LIN {X 0,Y 714.172,Z 1021.651,A -85,B 0,C 180,E1 33366.658,E2 33366.658} C_VEL
LIN {X 0,Y 714.698,Z 1002.417,A -85,B 0,C 180,E1 33365.36,E2 33365.36} C_VEL
LIN {X 0,Y 715.219,Z 981.551,A -85,B 0,C 180,E1 33364.139,E2 33364.139} C_VEL
LIN {X 0,Y 715.786,Z 960.973,A -85,B 0,C 180,E1 33363.089,E2 33363.089} C_VEL
LIN {X 0,Y 716.314,Z 937.723,A -85,B 0,C 180,E1 33362.08,E2 33362.08} C_VEL
LIN {X 0,Y 716.774,Z 917.131,A -85,B 0,C 180,E1 33361.323,E2 33361.323} C_VEL
LIN {X 0,Y 717.276,Z 891.994,A -85,B 0,C 180,E1 33360.566,E2 33360.566} C_VEL
LIN {X 0,Y 717.596,Z 870.583,A -85,B 0,C 180,E1 33360.057,E2 33360.057} C_VEL
LIN {X 0,Y 717.997,Z 845.408,A -85,B 0,C 180,E1 33359.611,E2 33359.611} C_VEL
LIN {X 0,Y 718.258,Z 792.779,A -85,B 0,C 180,E1 33358.994,E2 33358.994} C_VEL
LIN {X 0,Y 719.244,Z 571.123,A -85,B 0,C 180,E1 33356.478,E2 33356.478} C_VEL
LIN {X 0,Y 719.679,Z 463.116,A -85,B 0,C 180,E1 33355.225,E2 33355.225} C_VEL
LIN {X 0,Y 717.181,Z 452.735,A -85,B 0,C 180,E1 33354.942,E2 33354.942} C_VEL
LIN {X 0,Y 717.903,Z 418.681,A -85,B 0,C 180,E1 33352.551,E2 33352.551} C_VEL
LIN {X 0,Y 712.298,Z 403.677,A -85,B 0,C 180,E1 33351.077,E2 33351.077} C_VEL
LIN {X 0,Y 712.228,Z 403.51,A -85,B 0,C 180,E1 33348.283,E2 33348.283} C_VEL
LIN {X 0,Y 712.278,Z 403.505,A -85,B 0,C 180,E1 33345.42,E2 33345.42} C_VEL
LIN {X 0,Y 712.238,Z 403.496,A -85,B 0,C 180,E1 33342.475,E2 33342.475} C_VEL
LIN {X 0,Y 712.277,Z 403.502,A -85,B 0,C 180,E1 33339.584,E2 33339.584} C_VEL
LIN {X 0,Y 712.255,Z 403.497,A -85,B 0,C 180,E1 33336.529,E2 33336.529} C_VEL
LIN {X 0,Y 712.277,Z 403.507,A -85,B 0,C 180,E1 33333.58,E2 33333.58} C_VEL
LIN {X 0,Y 712.263,Z 403.501,A -85,B 0,C 180,E1 33330.464,E2 33330.464} C_VEL
LIN {X 0,Y 712.279,Z 403.507,A -85,B 0,C 180,E1 33327.476,E2 33327.476} C_VEL
LIN {X 0,Y 712.269,Z 403.495,A -85,B 0,C 180,E1 33324.376,E2 33324.376} C_VEL
LIN {X 0,Y 712.281,Z 403.51,A -85,B 0,C 180,E1 33321.407,E2 33321.407} C_VEL
LIN {X 0,Y 712.275,Z 403.495,A -85,B 0,C 180,E1 33318.328,E2 33318.328} C_VEL
LIN {X 0,Y 712.28,Z 403.504,A -85,B 0,C 180,E1 33315.302,E2 33315.302} C_VEL
LIN {X 0,Y 712.28,Z 403.498,A -85,B 0,C 180,E1 33312.238,E2 33312.238} C_VEL
LIN {X 0,Y 712.272,Z 403.502,A -85,B 0,C 180,E1 33309.209,E2 33309.209} C_VEL
LIN {X 0,Y 712.276,Z 403.499,A -85,B 0,C 180,E1 33306.205,E2 33306.205} C_VEL
LIN {X 0,Y 712.268,Z 403.504,A -85,B 0,C 180,E1 33303.138,E2 33303.138} C_VEL
LIN {X 0,Y 712.267,Z 403.5,A -85,B 0,C 180,E1 33300.161,E2 33300.161} C_VEL
LIN {X 0,Y 712.261,Z 403.507,A -85,B 0,C 180,E1 33297.023,E2 33297.023} C_VEL
LIN {X 0,Y 712.255,Z 403.501,A -85,B 0,C 180,E1 33294.118,E2 33294.118} C_VEL
LIN {X 0,Y 712.265,Z 403.508,A -85,B 0,C 180,E1 33291.035,E2 33291.035} C_VEL
LIN {X 0,Y 712.233,Z 403.504,A -85,B 0,C 180,E1 33288.255,E2 33288.255} C_VEL
LIN {X 0,Y 712.281,Z 403.501,A -85,B 0,C 180,E1 33285.288,E2 33285.288} C_VEL
LIN {X 0,Y 712.223,Z 403.504,A -85,B 0,C 180,E1 33282.432,E2 33282.432} C_VEL
LIN {X 0,Y 712.253,Z 403.506,A -85,B 0,C 180,E1 33280.882,E2 33280.882} C_VEL
LIN {X 0,Y 711.211,Z 403.637,A -85,B 0,C 180,E1 33280.262,E2 33280.262} C_VEL
LIN {X 0,Y 704.791,Z 404.436,A -85,B 0,C 180,E1 33278.526,E2 33278.526} C_VEL
LIN {X 0,Y 704.281,Z 404.495,A -85,B 0,C 180,E1 33278.075,E2 33278.075} C_VEL
LIN {X 0,Y 704.342,Z 404.49,A -85,B 0,C 180,E1 33275.152,E2 33275.152} C_VEL
LIN {X 0,Y 704.273,Z 404.493,A -85,B 0,C 180,E1 33272.338,E2 33272.338} C_VEL
LIN {X 0,Y 704.287,Z 404.495,A -85,B 0,C 180,E1 33269.735,E2 33269.735} C_VEL
LIN {X 0,Y 704.284,Z 404.499,A -85,B 0,C 180,E1 33266.574,E2 33266.574} C_VEL
LIN {X 0,Y 704.259,Z 404.496,A -85,B 0,C 180,E1 33264,E2 33264} C_VEL
LIN {X 0,Y 704.331,Z 404.496,A -85,B 0,C 180,E1 33261.204,E2 33261.204} C_VEL
LIN {X 0,Y 704.254,Z 404.476,A -85,B 0,C 180,E1 33258.25,E2 33258.25} C_VEL
LIN {X 0,Y 704.248,Z 404.498,A -85,B 0,C 180,E1 33255.803,E2 33255.803} C_VEL
LIN {X 0,Y 704.323,Z 404.484,A -85,B 0,C 180,E1 33253.019,E2 33253.019} C_VEL
LIN {X 0,Y 704.244,Z 404.504,A -85,B 0,C 180,E1 33250.135,E2 33250.135} C_VEL
LIN {X 0,Y 704.232,Z 404.493,A -85,B 0,C 180,E1 33247.834,E2 33247.834} C_VEL
LIN {X 0,Y 704.252,Z 404.503,A -85,B 0,C 180,E1 33245.4,E2 33245.4} C_VEL
LIN {X 0,Y 704.289,Z 404.785,A -85,B 0,C 180,E1 33243.45,E2 33243.45} C_VEL
LIN {X 0,Y 707.485,Z 413.87,A -85,B 0,C 180,E1 33242.537,E2 33242.537} C_VEL
LIN {X 0,Y 712.329,Z 423.155,A -85,B 0,C 180,E1 33242.141,E2 33242.141} C_VEL
LIN {X 0,Y 713.266,Z 427.659,A -85,B 0,C 180,E1 33242.033,E2 33242.033} C_VEL
LIN {X 0,Y 711.801,Z 678.151,A -85,B 0,C 180,E1 33239.141,E2 33239.141} C_VEL
LIN {X 0,Y 711.089,Z 803.093,A -85,B 0,C 180,E1 33237.703,E2 33237.703} C_VEL
LIN {X 0,Y 710.685,Z 828.598,A -85,B 0,C 180,E1 33237.264,E2 33237.264} C_VEL
LIN {X 0,Y 710.266,Z 850.477,A -85,B 0,C 180,E1 33236.75,E2 33236.75} C_VEL
LIN {X 0,Y 709.752,Z 874.703,A -85,B 0,C 180,E1 33236.03,E2 33236.03} C_VEL
LIN {X 0,Y 709.172,Z 896.162,A -85,B 0,C 180,E1 33235.246,E2 33235.246} C_VEL
LIN {X 0,Y 708.554,Z 919.316,A -85,B 0,C 180,E1 33234.246,E2 33234.246} C_VEL
LIN {X 0,Y 707.886,Z 940.548,A -85,B 0,C 180,E1 33233.161,E2 33233.161} C_VEL
LIN {X 0,Y 707.238,Z 961.765,A -85,B 0,C 180,E1 33231.916,E2 33231.916} C_VEL
LIN {X 0,Y 706.634,Z 980.711,A -85,B 0,C 180,E1 33230.63,E2 33230.63} C_VEL
LIN {X 0,Y 706.061,Z 999.843,A -85,B 0,C 180,E1 33229.165,E2 33229.165} C_VEL
LIN {X 0,Y 705.555,Z 1017.001,A -85,B 0,C 180,E1 33227.654,E2 33227.654} C_VEL
LIN {X 0,Y 705.105,Z 1033.94,A -85,B 0,C 180,E1 33225.968,E2 33225.968} C_VEL
LIN {X 0,Y 704.748,Z 1047.913,A -85,B 0,C 180,E1 33224.376,E2 33224.376} C_VEL
LIN {X 0,Y 704.478,Z 1062.037,A -85,B 0,C 180,E1 33222.542,E2 33222.542} C_VEL
LIN {X 0,Y 704.26,Z 1073.543,A -85,B 0,C 180,E1 33220.802,E2 33220.802} C_VEL
LIN {X 0,Y 704.097,Z 1084.379,A -85,B 0,C 180,E1 33218.905,E2 33218.905} C_VEL
LIN {X 0,Y 703.993,Z 1092.895,A -85,B 0,C 180,E1 33217.098,E2 33217.098} C_VEL
LIN {X 0,Y 703.942,Z 1099.381,A -85,B 0,C 180,E1 33215.461,E2 33215.461} C_VEL
LIN {X 0,Y 703.9,Z 1105.808,A -85,B 0,C 180,E1 33213.42,E2 33213.42} C_VEL
LIN {X 0,Y 703.919,Z 1109.758,A -85,B 0,C 180,E1 33211.709,E2 33211.709} C_VEL
LIN {X 0,Y 703.913,Z 1112.752,A -85,B 0,C 180,E1 33209.837,E2 33209.837} C_VEL
LIN {X 0,Y 703.905,Z 1114.275,A -85,B 0,C 180,E1 33207.802,E2 33207.802} C_VEL
LIN {X 0,Y 703.9,Z 1114.27,A -85,B 0,C 180,E1 33206.09,E2 33206.09} C_VEL
LIN {X 0,Y 703.913,Z 1112.605,A -85,B 0,C 180,E1 33203.966,E2 33203.966} C_VEL
LIN {X 0,Y 703.92,Z 1109.684,A -85,B 0,C 180,E1 33202.162,E2 33202.162} C_VEL
LIN {X 0,Y 703.92,Z 1105.02,A -85,B 0,C 180,E1 33200.186,E2 33200.186} C_VEL
LIN {X 0,Y 703.938,Z 1098.76,A -85,B 0,C 180,E1 33198.28,E2 33198.28} C_VEL
LIN {X 0,Y 704.017,Z 1092.046,A -85,B 0,C 180,E1 33196.614,E2 33196.614} C_VEL
LIN {X 0,Y 704.116,Z 1082.18,A -85,B 0,C 180,E1 33194.6,E2 33194.6} C_VEL
LIN {X 0,Y 704.27,Z 1072.308,A -85,B 0,C 180,E1 33192.909,E2 33192.909} C_VEL
LIN {X 0,Y 704.521,Z 1059.625,A -85,B 0,C 180,E1 33191.034,E2 33191.034} C_VEL
LIN {X 0,Y 704.777,Z 1046.795,A -85,B 0,C 180,E1 33189.4,E2 33189.4} C_VEL
LIN {X 0,Y 705.159,Z 1031.359,A -85,B 0,C 180,E1 33187.665,E2 33187.665} C_VEL
LIN {X 0,Y 705.585,Z 1015.693,A -85,B 0,C 180,E1 33186.135,E2 33186.135} C_VEL
LIN {X 0,Y 706.113,Z 997.953,A -85,B 0,C 180,E1 33184.592,E2 33184.592} C_VEL
LIN {X 0,Y 706.658,Z 980.061,A -85,B 0,C 180,E1 33183.233,E2 33183.233} C_VEL
LIN {X 0,Y 707.287,Z 959.785,A -85,B 0,C 180,E1 33181.87,E2 33181.87} C_VEL
LIN {X 0,Y 707.92,Z 939.612,A -85,B 0,C 180,E1 33180.698,E2 33180.698} C_VEL
LIN {X 0,Y 708.605,Z 917.18,A -85,B 0,C 180,E1 33179.564,E2 33179.564} C_VEL
LIN {X 0,Y 709.184,Z 895.817,A -85,B 0,C 180,E1 33178.65,E2 33178.65} C_VEL
LIN {X 0,Y 709.806,Z 873.141,A -85,B 0,C 180,E1 33177.827,E2 33177.827} C_VEL
LIN {X 0,Y 710.287,Z 849.001,A -85,B 0,C 180,E1 33177.122,E2 33177.122} C_VEL
LIN {X 0,Y 710.771,Z 825.796,A -85,B 0,C 180,E1 33176.587,E2 33176.587} C_VEL
LIN {X 0,Y 711.1,Z 801.196,A -85,B 0,C 180,E1 33176.182,E2 33176.182} C_VEL
LIN {X 0,Y 712.566,Z 543.422,A -85,B 0,C 180,E1 33173.223,E2 33173.223} C_VEL
LIN {X 0,Y 713.097,Z 426.002,A -85,B 0,C 180,E1 33171.847,E2 33171.847} C_VEL
LIN {X 0,Y 711.559,Z 421.352,A -85,B 0,C 180,E1 33171.704,E2 33171.704} C_VEL
LIN {X 0,Y 707.344,Z 413.486,A -85,B 0,C 180,E1 33171.347,E2 33171.347} C_VEL
LIN {X 0,Y 704.271,Z 404.702,A -85,B 0,C 180,E1 33170.437,E2 33170.437} C_VEL
LIN {X 0,Y 704.236,Z 404.507,A -85,B 0,C 180,E1 33168.073,E2 33168.073} C_VEL
LIN {X 0,Y 704.276,Z 404.505,A -85,B 0,C 180,E1 33165.464,E2 33165.464} C_VEL
LIN {X 0,Y 704.262,Z 404.486,A -85,B 0,C 180,E1 33162.407,E2 33162.407} C_VEL
LIN {X 0,Y 704.249,Z 404.498,A -85,B 0,C 180,E1 33159.923,E2 33159.923} C_VEL
LIN {X 0,Y 704.28,Z 404.497,A -85,B 0,C 180,E1 33157.42,E2 33157.42} C_VEL
LIN {X 0,Y 704.275,Z 404.496,A -85,B 0,C 180,E1 33154.28,E2 33154.28} C_VEL
LIN {X 0,Y 704.262,Z 404.497,A -85,B 0,C 180,E1 33151.74,E2 33151.74} C_VEL
LIN {X 0,Y 704.339,Z 404.476,A -85,B 0,C 180,E1 33148.953,E2 33148.953} C_VEL
LIN {X 0,Y 704.277,Z 404.496,A -85,B 0,C 180,E1 33146.012,E2 33146.012} C_VEL
LIN {X 0,Y 704.282,Z 404.493,A -85,B 0,C 180,E1 33143.424,E2 33143.424} C_VEL
LIN {X 0,Y 704.337,Z 404.487,A -85,B 0,C 180,E1 33140.44,E2 33140.44} C_VEL
LIN {X 0,Y 704.281,Z 404.497,A -85,B 0,C 180,E1 33137.602,E2 33137.602} C_VEL
LIN {X 0,Y 704.346,Z 404.494,A -85,B 0,C 180,E1 33134.805,E2 33134.805} C_VEL
LIN {X 0,Y 704.296,Z 404.488,A -85,B 0,C 180,E1 33131.797,E2 33131.797} C_VEL
LIN {X 0,Y 704.321,Z 404.499,A -85,B 0,C 180,E1 33128.984,E2 33128.984} C_VEL
LIN {X 0,Y 704.314,Z 404.488,A -85,B 0,C 180,E1 33125.867,E2 33125.867} C_VEL
LIN {X 0,Y 704.324,Z 404.498,A -85,B 0,C 180,E1 33122.93,E2 33122.93} C_VEL
LIN {X 0,Y 704.327,Z 404.489,A -85,B 0,C 180,E1 33119.837,E2 33119.837} C_VEL
LIN {X 0,Y 704.33,Z 404.491,A -85,B 0,C 180,E1 33116.826,E2 33116.826} C_VEL
LIN {X 0,Y 704.331,Z 404.486,A -85,B 0,C 180,E1 33113.724,E2 33113.724} C_VEL
LIN {X 0,Y 704.337,Z 404.497,A -85,B 0,C 180,E1 33110.686,E2 33110.686} C_VEL
LIN {X 0,Y 704.334,Z 404.482,A -85,B 0,C 180,E1 33107.609,E2 33107.609} C_VEL
LIN {X 0,Y 704.34,Z 404.494,A -85,B 0,C 180,E1 33104.521,E2 33104.521} C_VEL
LIN {X 0,Y 704.334,Z 404.489,A -85,B 0,C 180,E1 33101.458,E2 33101.458} C_VEL
LIN {X 0,Y 704.333,Z 404.488,A -85,B 0,C 180,E1 33098.413,E2 33098.413} C_VEL
LIN {X 0,Y 704.342,Z 404.488,A -85,B 0,C 180,E1 33095.421,E2 33095.421} C_VEL
LIN {X 0,Y 704.328,Z 404.495,A -85,B 0,C 180,E1 33092.34,E2 33092.34} C_VEL
LIN {X 0,Y 704.34,Z 404.485,A -85,B 0,C 180,E1 33089.349,E2 33089.349} C_VEL
LIN {X 0,Y 704.327,Z 404.497,A -85,B 0,C 180,E1 33086.284,E2 33086.284} C_VEL
LIN {X 0,Y 704.332,Z 404.489,A -85,B 0,C 180,E1 33083.297,E2 33083.297} C_VEL
LIN {X 0,Y 704.317,Z 404.497,A -85,B 0,C 180,E1 33080.178,E2 33080.178} C_VEL
LIN {X 0,Y 704.318,Z 404.486,A -85,B 0,C 180,E1 33077.266,E2 33077.266} C_VEL
LIN {X 0,Y 704.321,Z 404.495,A -85,B 0,C 180,E1 33074.191,E2 33074.191} C_VEL
LIN {X 0,Y 704.296,Z 404.499,A -85,B 0,C 180,E1 33071.421,E2 33071.421} C_VEL
LIN {X 0,Y 704.325,Z 404.718,A -85,B 0,C 180,E1 33069.336,E2 33069.336} C_VEL
LIN {X 0,Y 710.956,Z 422.229,A -85,B 0,C 180,E1 33067.617,E2 33067.617} C_VEL
LIN {X 0,Y 710.223,Z 453.298,A -85,B 0,C 180,E1 33065.43,E2 33065.43} C_VEL
LIN {X 0,Y 713.265,Z 466.404,A -85,B 0,C 180,E1 33065.094,E2 33065.094} C_VEL
LIN {X 0,Y 711.805,Z 716.052,A -85,B 0,C 180,E1 33062.21,E2 33062.21} C_VEL
LIN {X 0,Y 711.1,Z 842.987,A -85,B 0,C 180,E1 33060.749,E2 33060.749} C_VEL
LIN {X 0,Y 710.684,Z 868.493,A -85,B 0,C 180,E1 33060.311,E2 33060.311} C_VEL
LIN {X 0,Y 710.261,Z 890.337,A -85,B 0,C 180,E1 33059.798,E2 33059.798} C_VEL
LIN {X 0,Y 709.761,Z 914.559,A -85,B 0,C 180,E1 33059.08,E2 33059.08} C_VEL
LIN {X 0,Y 709.162,Z 936.485,A -85,B 0,C 180,E1 33058.278,E2 33058.278} C_VEL
LIN {X 0,Y 708.561,Z 959.167,A -85,B 0,C 180,E1 33057.299,E2 33057.299} C_VEL
LIN {X 0,Y 707.877,Z 980.757,A -85,B 0,C 180,E1 33056.194,E2 33056.194} C_VEL
LIN {X 0,Y 707.237,Z 1001.75,A -85,B 0,C 180,E1 33054.962,E2 33054.962} C_VEL
LIN {X 0,Y 706.629,Z 1021.05,A -85,B 0,C 180,E1 33053.651,E2 33053.651} C_VEL
LIN {X 0,Y 706.064,Z 1039.761,A -85,B 0,C 180,E1 33052.217,E2 33052.217} C_VEL
LIN {X 0,Y 705.561,Z 1056.796,A -85,B 0,C 180,E1 33050.719,E2 33050.719} C_VEL
LIN {X 0,Y 705.139,Z 1072.966,A -85,B 0,C 180,E1 33049.121,E2 33049.121} C_VEL
LIN {X 0,Y 704.764,Z 1087.223,A -85,B 0,C 180,E1 33047.504,E2 33047.504} C_VEL
LIN {X 0,Y 704.491,Z 1101.06,A -85,B 0,C 180,E1 33045.729,E2 33045.729} C_VEL
LIN {X 0,Y 704.27,Z 1112.797,A -85,B 0,C 180,E1 33043.967,E2 33043.967} C_VEL
LIN {X 0,Y 704.122,Z 1122.947,A -85,B 0,C 180,E1 33042.215,E2 33042.215} C_VEL
LIN {X 0,Y 704.014,Z 1132.538,A -85,B 0,C 180,E1 33040.226,E2 33040.226} C_VEL
LIN {X 0,Y 703.947,Z 1139.12,A -85,B 0,C 180,E1 33038.577,E2 33038.577} C_VEL
LIN {X 0,Y 703.922,Z 1145.451,A -85,B 0,C 180,E1 33036.607,E2 33036.607} C_VEL
LIN {X 0,Y 703.911,Z 1149.814,A -85,B 0,C 180,E1 33034.726,E2 33034.726} C_VEL
LIN {X 0,Y 703.882,Z 1152.685,A -85,B 0,C 180,E1 33032.931,E2 33032.931} C_VEL
LIN {X 0,Y 703.892,Z 1154.262,A -85,B 0,C 180,E1 33030.895,E2 33030.895} C_VEL
LIN {X 0,Y 703.884,Z 1154.306,A -85,B 0,C 180,E1 33029.267,E2 33029.267} C_VEL
LIN {X 0,Y 703.886,Z 1153.017,A -85,B 0,C 180,E1 33027.313,E2 33027.313} C_VEL
LIN {X 0,Y 703.916,Z 1149.972,A -85,B 0,C 180,E1 33025.356,E2 33025.356} C_VEL
LIN {X 0,Y 703.921,Z 1145.864,A -85,B 0,C 180,E1 33023.557,E2 33023.557} C_VEL
LIN {X 0,Y 703.948,Z 1139.423,A -85,B 0,C 180,E1 33021.505,E2 33021.505} C_VEL
LIN {X 0,Y 704.009,Z 1132.739,A -85,B 0,C 180,E1 33019.821,E2 33019.821} C_VEL
LIN {X 0,Y 704.116,Z 1123.406,A -85,B 0,C 180,E1 33017.868,E2 33017.868} C_VEL
LIN {X 0,Y 704.262,Z 1113.319,A -85,B 0,C 180,E1 33016.117,E2 33016.117} C_VEL
LIN {X 0,Y 704.473,Z 1101.643,A -85,B 0,C 180,E1 33014.355,E2 33014.355} C_VEL
LIN {X 0,Y 704.746,Z 1087.93,A -85,B 0,C 180,E1 33012.58,E2 33012.58} C_VEL
LIN {X 0,Y 705.118,Z 1073.742,A -85,B 0,C 180,E1 33010.965,E2 33010.965} C_VEL
LIN {X 0,Y 705.542,Z 1057.389,A -85,B 0,C 180,E1 33009.336,E2 33009.336} C_VEL
LIN {X 0,Y 706.035,Z 1040.55,A -85,B 0,C 180,E1 33007.85,E2 33007.85} C_VEL
LIN {X 0,Y 706.609,Z 1021.653,A -85,B 0,C 180,E1 33006.393,E2 33006.393} C_VEL
LIN {X 0,Y 707.213,Z 1002.413,A -85,B 0,C 180,E1 33005.082,E2 33005.082} C_VEL
LIN {X 0,Y 707.847,Z 981.555,A -85,B 0,C 180,E1 33003.85,E2 33003.85} C_VEL
LIN {X 0,Y 708.499,Z 960.969,A -85,B 0,C 180,E1 33002.79,E2 33002.79} C_VEL
LIN {X 0,Y 709.128,Z 937.608,A -85,B 0,C 180,E1 33001.766,E2 33001.766} C_VEL
LIN {X 0,Y 709.672,Z 917.128,A -85,B 0,C 180,E1 33001.008,E2 33001.008} C_VEL
LIN {X 0,Y 710.244,Z 892.062,A -85,B 0,C 180,E1 33000.247,E2 33000.247} C_VEL
LIN {X 0,Y 710.629,Z 870.451,A -85,B 0,C 180,E1 32999.73,E2 32999.73} C_VEL
LIN {X 0,Y 711.088,Z 845.088,A -85,B 0,C 180,E1 32999.28,E2 32999.28} C_VEL
LIN {X 0,Y 711.421,Z 788.58,A -85,B 0,C 180,E1 32998.614,E2 32998.614} C_VEL
LIN {X 0,Y 712.582,Z 568.705,A -85,B 0,C 180,E1 32996.094,E2 32996.094} C_VEL
LIN {X 0,Y 713.087,Z 464.856,A -85,B 0,C 180,E1 32994.878,E2 32994.878} C_VEL
LIN {X 0,Y 710.17,Z 452.741,A -85,B 0,C 180,E1 32994.544,E2 32994.544} C_VEL
LIN {X 0,Y 710.885,Z 422.01,A -85,B 0,C 180,E1 32992.362,E2 32992.362} C_VEL
LIN {X 0,Y 704.321,Z 404.695,A -85,B 0,C 180,E1 32990.653,E2 32990.653} C_VEL
LIN {X 0,Y 704.3,Z 404.496,A -85,B 0,C 180,E1 32988.035,E2 32988.035} C_VEL
LIN {X 0,Y 704.34,Z 404.492,A -85,B 0,C 180,E1 32984.989,E2 32984.989} C_VEL
LIN {X 0,Y 704.3,Z 404.478,A -85,B 0,C 180,E1 32982.075,E2 32982.075} C_VEL
LIN {X 0,Y 704.336,Z 404.495,A -85,B 0,C 180,E1 32979.178,E2 32979.178} C_VEL
LIN {X 0,Y 704.303,Z 404.489,A -85,B 0,C 180,E1 32976.256,E2 32976.256} C_VEL
LIN {X 0,Y 704.339,Z 404.492,A -85,B 0,C 180,E1 32973.411,E2 32973.411} C_VEL
LIN {X 0,Y 704.318,Z 404.492,A -85,B 0,C 180,E1 32970.358,E2 32970.358} C_VEL
LIN {X 0,Y 704.338,Z 404.497,A -85,B 0,C 180,E1 32967.384,E2 32967.384} C_VEL
LIN {X 0,Y 704.325,Z 404.484,A -85,B 0,C 180,E1 32964.312,E2 32964.312} C_VEL
LIN {X 0,Y 704.337,Z 404.497,A -85,B 0,C 180,E1 32961.311,E2 32961.311} C_VEL
LIN {X 0,Y 704.332,Z 404.485,A -85,B 0,C 180,E1 32958.243,E2 32958.243} C_VEL
LIN {X 0,Y 704.333,Z 404.492,A -85,B 0,C 180,E1 32955.226,E2 32955.226} C_VEL
LIN {X 0,Y 704.339,Z 404.487,A -85,B 0,C 180,E1 32952.212,E2 32952.212} C_VEL
LIN {X 0,Y 704.329,Z 404.49,A -85,B 0,C 180,E1 32949.149,E2 32949.149} C_VEL
LIN {X 0,Y 704.342,Z 404.488,A -85,B 0,C 180,E1 32946.112,E2 32946.112} C_VEL
LIN {X 0,Y 704.319,Z 404.493,A -85,B 0,C 180,E1 32943.011,E2 32943.011} C_VEL
LIN {X 0,Y 704.347,Z 404.488,A -85,B 0,C 180,E1 32940,E2 32940} C_VEL
LIN {X 0,Y 704.312,Z 404.494,A -85,B 0,C 180,E1 32936.908,E2 32936.908} C_VEL
LIN {X 0,Y 704.332,Z 404.489,A -85,B 0,C 180,E1 32933.97,E2 32933.97} C_VEL
LIN {X 0,Y 704.315,Z 404.497,A -85,B 0,C 180,E1 32930.933,E2 32930.933} C_VEL
LIN {X 0,Y 704.302,Z 404.491,A -85,B 0,C 180,E1 32928.12,E2 32928.12} C_VEL
LIN {X 0,Y 704.338,Z 404.494,A -85,B 0,C 180,E1 32925.111,E2 32925.111} C_VEL
LIN {X 0,Y 704.284,Z 404.492,A -85,B 0,C 180,E1 32922.296,E2 32922.296} C_VEL
LIN {X 0,Y 704.343,Z 404.49,A -85,B 0,C 180,E1 32919.386,E2 32919.386} C_VEL
LIN {X 0,Y 704.281,Z 404.495,A -85,B 0,C 180,E1 32918.075,E2 32918.075} C_VEL
LIN {X 0,Y 703.324,Z 404.621,A -85,B 0,C 180,E1 32917.448,E2 32917.448} C_VEL
LIN {X 0,Y 696.939,Z 405.403,A -85,B 0,C 180,E1 32915.692,E2 32915.692} C_VEL
LIN {X 0,Y 696.404,Z 405.475,A -85,B 0,C 180,E1 32915.236,E2 32915.236} C_VEL
LIN {X 0,Y 696.335,Z 405.482,A -85,B 0,C 180,E1 32912.367,E2 32912.367} C_VEL
LIN {X 0,Y 696.349,Z 405.484,A -85,B 0,C 180,E1 32909.735,E2 32909.735} C_VEL
LIN {X 0,Y 696.353,Z 405.488,A -85,B 0,C 180,E1 32906.636,E2 32906.636} C_VEL
LIN {X 0,Y 696.319,Z 405.485,A -85,B 0,C 180,E1 32904.033,E2 32904.033} C_VEL
LIN {X 0,Y 696.37,Z 405.486,A -85,B 0,C 180,E1 32901.347,E2 32901.347} C_VEL
LIN {X 0,Y 696.32,Z 405.462,A -85,B 0,C 180,E1 32898.329,E2 32898.329} C_VEL
LIN {X 0,Y 696.308,Z 405.487,A -85,B 0,C 180,E1 32895.856,E2 32895.856} C_VEL
LIN {X 0,Y 696.37,Z 405.474,A -85,B 0,C 180,E1 32893.116,E2 32893.116} C_VEL
LIN {X 0,Y 696.306,Z 405.493,A -85,B 0,C 180,E1 32890.148,E2 32890.148} C_VEL
LIN {X 0,Y 696.294,Z 405.481,A -85,B 0,C 180,E1 32887.82,E2 32887.82} C_VEL
LIN {X 0,Y 696.327,Z 405.486,A -85,B 0,C 180,E1 32885.258,E2 32885.258} C_VEL
LIN {X 0,Y 696.337,Z 405.747,A -85,B 0,C 180,E1 32883.883,E2 32883.883} C_VEL
LIN {X 0,Y 699.249,Z 413.816,A -85,B 0,C 180,E1 32883.026,E2 32883.026} C_VEL
LIN {X 0,Y 706.323,Z 427.111,A -85,B 0,C 180,E1 32882.437,E2 32882.437} C_VEL
LIN {X 0,Y 706.698,Z 430.076,A -85,B 0,C 180,E1 32882.379,E2 32882.379} C_VEL
LIN {X 0,Y 705.014,Z 680.25,A -85,B 0,C 180,E1 32879.464,E2 32879.464} C_VEL
LIN {X 0,Y 704.203,Z 803.228,A -85,B 0,C 180,E1 32878.035,E2 32878.035} C_VEL
LIN {X 0,Y 703.751,Z 828.68,A -85,B 0,C 180,E1 32877.593,E2 32877.593} C_VEL
LIN {X 0,Y 703.261,Z 850.534,A -85,B 0,C 180,E1 32877.076,E2 32877.076} C_VEL
LIN {X 0,Y 702.637,Z 875.784,A -85,B 0,C 180,E1 32876.314,E2 32876.314} C_VEL
LIN {X 0,Y 702.023,Z 896.009,A -85,B 0,C 180,E1 32875.567,E2 32875.567} C_VEL
LIN {X 0,Y 701.322,Z 918.305,A -85,B 0,C 180,E1 32874.602,E2 32874.602} C_VEL
LIN {X 0,Y 700.544,Z 940.37,A -85,B 0,C 180,E1 32873.467,E2 32873.467} C_VEL
LIN {X 0,Y 699.805,Z 961.02,A -85,B 0,C 180,E1 32872.249,E2 32872.249} C_VEL
LIN {X 0,Y 699.096,Z 980.58,A -85,B 0,C 180,E1 32870.911,E2 32870.911} C_VEL
LIN {X 0,Y 698.424,Z 999.594,A -85,B 0,C 180,E1 32869.442,E2 32869.442} C_VEL
LIN {X 0,Y 697.842,Z 1016.566,A -85,B 0,C 180,E1 32867.935,E2 32867.935} C_VEL
LIN {X 0,Y 697.336,Z 1032.748,A -85,B 0,C 180,E1 32866.322,E2 32866.322} C_VEL
LIN {X 0,Y 696.914,Z 1047.521,A -85,B 0,C 180,E1 32864.626,E2 32864.626} C_VEL
LIN {X 0,Y 696.6,Z 1061.144,A -85,B 0,C 180,E1 32862.855,E2 32862.855} C_VEL
LIN {X 0,Y 696.32,Z 1073.254,A -85,B 0,C 180,E1 32861.01,E2 32861.01} C_VEL
LIN {X 0,Y 696.137,Z 1083.703,A -85,B 0,C 180,E1 32859.174,E2 32859.174} C_VEL
LIN {X 0,Y 696.026,Z 1092.695,A -85,B 0,C 180,E1 32857.263,E2 32857.263} C_VEL
LIN {X 0,Y 695.948,Z 1099.51,A -85,B 0,C 180,E1 32855.524,E2 32855.524} C_VEL
LIN {X 0,Y 695.903,Z 1105.896,A -85,B 0,C 180,E1 32853.46,E2 32853.46} C_VEL
LIN {X 0,Y 695.92,Z 1109.826,A -85,B 0,C 180,E1 32851.729,E2 32851.729} C_VEL
LIN {X 0,Y 695.909,Z 1112.912,A -85,B 0,C 180,E1 32849.753,E2 32849.753} C_VEL
LIN {X 0,Y 695.903,Z 1114.284,A -85,B 0,C 180,E1 32847.777,E2 32847.777} C_VEL
LIN {X 0,Y 695.904,Z 1114.261,A -85,B 0,C 180,E1 32846.045,E2 32846.045} C_VEL
LIN {X 0,Y 695.918,Z 1112.558,A -85,B 0,C 180,E1 32843.897,E2 32843.897} C_VEL
LIN {X 0,Y 695.919,Z 1109.617,A -85,B 0,C 180,E1 32842.072,E2 32842.072} C_VEL
LIN {X 0,Y 695.933,Z 1104.911,A -85,B 0,C 180,E1 32840.072,E2 32840.072} C_VEL
LIN {X 0,Y 695.947,Z 1098.935,A -85,B 0,C 180,E1 32838.228,E2 32838.228} C_VEL
LIN {X 0,Y 696.039,Z 1092.251,A -85,B 0,C 180,E1 32836.543,E2 32836.543} C_VEL
LIN {X 0,Y 696.155,Z 1082.443,A -85,B 0,C 180,E1 32834.505,E2 32834.505} C_VEL
LIN {X 0,Y 696.329,Z 1072.607,A -85,B 0,C 180,E1 32832.794,E2 32832.794} C_VEL
LIN {X 0,Y 696.609,Z 1059.988,A -85,B 0,C 180,E1 32830.897,E2 32830.897} C_VEL
LIN {X 0,Y 696.923,Z 1047.201,A -85,B 0,C 180,E1 32829.245,E2 32829.245} C_VEL
LIN {X 0,Y 697.36,Z 1031.842,A -85,B 0,C 180,E1 32827.491,E2 32827.491} C_VEL
LIN {X 0,Y 697.873,Z 1015.528,A -85,B 0,C 180,E1 32825.878,E2 32825.878} C_VEL
LIN {X 0,Y 698.487,Z 997.829,A -85,B 0,C 180,E1 32824.324,E2 32824.324} C_VEL
LIN {X 0,Y 699.119,Z 979.873,A -85,B 0,C 180,E1 32822.947,E2 32822.947} C_VEL
LIN {X 0,Y 699.84,Z 959.882,A -85,B 0,C 180,E1 32821.59,E2 32821.59} C_VEL
LIN {X 0,Y 700.568,Z 939.715,A -85,B 0,C 180,E1 32820.407,E2 32820.407} C_VEL
LIN {X 0,Y 701.338,Z 917.756,A -85,B 0,C 180,E1 32819.282,E2 32819.282} C_VEL
LIN {X 0,Y 702.025,Z 895.969,A -85,B 0,C 180,E1 32818.342,E2 32818.342} C_VEL
LIN {X 0,Y 702.693,Z 874.286,A -85,B 0,C 180,E1 32817.545,E2 32817.545} C_VEL
LIN {X 0,Y 703.275,Z 849.84,A -85,B 0,C 180,E1 32816.816,E2 32816.816} C_VEL
LIN {X 0,Y 703.787,Z 827.578,A -85,B 0,C 180,E1 32816.294,E2 32816.294} C_VEL
LIN {X 0,Y 704.21,Z 802.207,A -85,B 0,C 180,E1 32815.861,E2 32815.861} C_VEL
LIN {X 0,Y 705.874,Z 548.474,A -85,B 0,C 180,E1 32812.92,E2 32812.92} C_VEL
LIN {X 0,Y 706.516,Z 427.832,A -85,B 0,C 180,E1 32811.493,E2 32811.493} C_VEL
LIN {X 0,Y 705.1,Z 424.445,A -85,B 0,C 180,E1 32811.37,E2 32811.37} C_VEL
LIN {X 0,Y 699.209,Z 413.723,A -85,B 0,C 180,E1 32810.877,E2 32810.877} C_VEL
LIN {X 0,Y 696.341,Z 405.812,A -85,B 0,C 180,E1 32810.043,E2 32810.043} C_VEL
LIN {X 0,Y 696.384,Z 405.476,A -85,B 0,C 180,E1 32809.173,E2 32809.173} C_VEL
LIN {X 0,Y 696.304,Z 405.494,A -85,B 0,C 180,E1 32806.246,E2 32806.246} C_VEL
LIN {X 0,Y 696.31,Z 405.493,A -85,B 0,C 180,E1 32803.8,E2 32803.8} C_VEL
LIN {X 0,Y 696.394,Z 405.468,A -85,B 0,C 180,E1 32800.899,E2 32800.899} C_VEL
LIN {X 0,Y 696.316,Z 405.487,A -85,B 0,C 180,E1 32798.102,E2 32798.102} C_VEL
LIN {X 0,Y 696.321,Z 405.462,A -85,B 0,C 180,E1 32795.634,E2 32795.634} C_VEL
LIN {X 0,Y 696.392,Z 405.483,A -85,B 0,C 180,E1 32792.675,E2 32792.675} C_VEL
LIN {X 0,Y 696.323,Z 405.463,A -85,B 0,C 180,E1 32789.886,E2 32789.886} C_VEL
LIN {X 0,Y 696.357,Z 405.482,A -85,B 0,C 180,E1 32787.261,E2 32787.261} C_VEL
LIN {X 0,Y 696.354,Z 405.478,A -85,B 0,C 180,E1 32784.157,E2 32784.157} C_VEL
LIN {X 0,Y 696.34,Z 405.487,A -85,B 0,C 180,E1 32781.49,E2 32781.49} C_VEL
LIN {X 0,Y 696.405,Z 405.484,A -85,B 0,C 180,E1 32778.587,E2 32778.587} C_VEL
LIN {X 0,Y 696.344,Z 405.477,A -85,B 0,C 180,E1 32775.662,E2 32775.662} C_VEL
LIN {X 0,Y 696.397,Z 405.486,A -85,B 0,C 180,E1 32772.859,E2 32772.859} C_VEL
LIN {X 0,Y 696.364,Z 405.481,A -85,B 0,C 180,E1 32769.838,E2 32769.838} C_VEL
LIN {X 0,Y 696.377,Z 405.484,A -85,B 0,C 180,E1 32767.01,E2 32767.01} C_VEL
LIN {X 0,Y 696.381,Z 405.479,A -85,B 0,C 180,E1 32763.87,E2 32763.87} C_VEL
LIN {X 0,Y 696.386,Z 405.48,A -85,B 0,C 180,E1 32760.905,E2 32760.905} C_VEL
LIN {X 0,Y 696.386,Z 405.472,A -85,B 0,C 180,E1 32757.778,E2 32757.778} C_VEL
LIN {X 0,Y 696.399,Z 405.487,A -85,B 0,C 180,E1 32754.728,E2 32754.728} C_VEL
LIN {X 0,Y 696.387,Z 405.474,A -85,B 0,C 180,E1 32751.606,E2 32751.606} C_VEL
LIN {X 0,Y 696.398,Z 405.48,A -85,B 0,C 180,E1 32748.572,E2 32748.572} C_VEL
LIN {X 0,Y 696.395,Z 405.478,A -85,B 0,C 180,E1 32745.532,E2 32745.532} C_VEL
LIN {X 0,Y 696.396,Z 405.485,A -85,B 0,C 180,E1 32742.436,E2 32742.436} C_VEL
LIN {X 0,Y 696.395,Z 405.475,A -85,B 0,C 180,E1 32739.404,E2 32739.404} C_VEL
LIN {X 0,Y 696.392,Z 405.488,A -85,B 0,C 180,E1 32736.356,E2 32736.356} C_VEL
LIN {X 0,Y 696.398,Z 405.469,A -85,B 0,C 180,E1 32733.294,E2 32733.294} C_VEL
LIN {X 0,Y 696.387,Z 405.484,A -85,B 0,C 180,E1 32730.305,E2 32730.305} C_VEL
LIN {X 0,Y 696.401,Z 405.477,A -85,B 0,C 180,E1 32727.286,E2 32727.286} C_VEL
LIN {X 0,Y 696.381,Z 405.482,A -85,B 0,C 180,E1 32724.219,E2 32724.219} C_VEL
LIN {X 0,Y 696.397,Z 405.476,A -85,B 0,C 180,E1 32721.228,E2 32721.228} C_VEL
LIN {X 0,Y 696.374,Z 405.48,A -85,B 0,C 180,E1 32718.112,E2 32718.112} C_VEL
LIN {X 0,Y 696.384,Z 405.481,A -85,B 0,C 180,E1 32715.178,E2 32715.178} C_VEL
LIN {X 0,Y 696.37,Z 405.48,A -85,B 0,C 180,E1 32712.069,E2 32712.069} C_VEL
LIN {X 0,Y 696.382,Z 405.718,A -85,B 0,C 180,E1 32709.769,E2 32709.769} C_VEL
LIN {X 0,Y 703.924,Z 425.709,A -85,B 0,C 180,E1 32707.785,E2 32707.785} C_VEL
LIN {X 0,Y 703.199,Z 452.864,A -85,B 0,C 180,E1 32705.856,E2 32705.856} C_VEL
LIN {X 0,Y 706.699,Z 468.246,A -85,B 0,C 180,E1 32705.446,E2 32705.446} C_VEL
LIN {X 0,Y 705.026,Z 717.07,A -85,B 0,C 180,E1 32702.546,E2 32702.546} C_VEL
LIN {X 0,Y 704.214,Z 843.106,A -85,B 0,C 180,E1 32701.081,E2 32701.081} C_VEL
LIN {X 0,Y 703.75,Z 868.622,A -85,B 0,C 180,E1 32700.639,E2 32700.639} C_VEL
LIN {X 0,Y 703.255,Z 890.448,A -85,B 0,C 180,E1 32700.123,E2 32700.123} C_VEL
LIN {X 0,Y 702.685,Z 914.555,A -85,B 0,C 180,E1 32699.401,E2 32699.401} C_VEL
LIN {X 0,Y 702.046,Z 935.354,A -85,B 0,C 180,E1 32698.637,E2 32698.637} C_VEL
LIN {X 0,Y 701.345,Z 957.243,A -85,B 0,C 180,E1 32697.696,E2 32697.696} C_VEL
LIN {X 0,Y 700.588,Z 979.137,A -85,B 0,C 180,E1 32696.579,E2 32696.579} C_VEL
LIN {X 0,Y 699.875,Z 998.827,A -85,B 0,C 180,E1 32695.429,E2 32695.429} C_VEL
LIN {X 0,Y 699.143,Z 1019.23,A -85,B 0,C 180,E1 32694.054,E2 32694.054} C_VEL
LIN {X 0,Y 698.498,Z 1037.255,A -85,B 0,C 180,E1 32692.676,E2 32692.676} C_VEL
LIN {X 0,Y 697.905,Z 1054.847,A -85,B 0,C 180,E1 32691.141,E2 32691.141} C_VEL
LIN {X 0,Y 697.405,Z 1070.484,A -85,B 0,C 180,E1 32689.603,E2 32689.603} C_VEL
LIN {X 0,Y 696.969,Z 1085.81,A -85,B 0,C 180,E1 32687.879,E2 32687.879} C_VEL
LIN {X 0,Y 696.63,Z 1098.842,A -85,B 0,C 180,E1 32686.212,E2 32686.212} C_VEL
LIN {X 0,Y 696.35,Z 1112.069,A -85,B 0,C 180,E1 32684.248,E2 32684.248} C_VEL
LIN {X 0,Y 696.181,Z 1122.028,A -85,B 0,C 180,E1 32682.526,E2 32682.526} C_VEL
LIN {X 0,Y 696.046,Z 1132.184,A -85,B 0,C 180,E1 32680.428,E2 32680.428} C_VEL
LIN {X 0,Y 695.952,Z 1139.003,A -85,B 0,C 180,E1 32678.709,E2 32678.709} C_VEL
LIN {X 0,Y 695.932,Z 1145.244,A -85,B 0,C 180,E1 32676.766,E2 32676.766} C_VEL
LIN {X 0,Y 695.906,Z 1149.814,A -85,B 0,C 180,E1 32674.78,E2 32674.78} C_VEL
LIN {X 0,Y 695.883,Z 1152.685,A -85,B 0,C 180,E1 32672.965,E2 32672.965} C_VEL
LIN {X 0,Y 695.893,Z 1154.262,A -85,B 0,C 180,E1 32670.906,E2 32670.906} C_VEL
LIN {X 0,Y 695.885,Z 1154.306,A -85,B 0,C 180,E1 32669.259,E2 32669.259} C_VEL
LIN {X 0,Y 695.885,Z 1153.017,A -85,B 0,C 180,E1 32667.282,E2 32667.282} C_VEL
LIN {X 0,Y 695.917,Z 1150.131,A -85,B 0,C 180,E1 32665.385,E2 32665.385} C_VEL
LIN {X 0,Y 695.925,Z 1146.277,A -85,B 0,C 180,E1 32663.648,E2 32663.648} C_VEL
LIN {X 0,Y 695.959,Z 1140.029,A -85,B 0,C 180,E1 32661.573,E2 32661.573} C_VEL
LIN {X 0,Y 696.021,Z 1133.249,A -85,B 0,C 180,E1 32659.822,E2 32659.822} C_VEL
LIN {X 0,Y 696.135,Z 1124.707,A -85,B 0,C 180,E1 32657.979,E2 32657.979} C_VEL
LIN {X 0,Y 696.316,Z 1113.84,A -85,B 0,C 180,E1 32656.04,E2 32656.04} C_VEL
LIN {X 0,Y 696.539,Z 1102.803,A -85,B 0,C 180,E1 32654.343,E2 32654.343} C_VEL
LIN {X 0,Y 696.878,Z 1088.633,A -85,B 0,C 180,E1 32652.464,E2 32652.464} C_VEL
LIN {X 0,Y 697.294,Z 1074.521,A -85,B 0,C 180,E1 32650.83,E2 32650.83} C_VEL
LIN {X 0,Y 697.821,Z 1057.388,A -85,B 0,C 180,E1 32649.097,E2 32649.097} C_VEL
LIN {X 0,Y 698.378,Z 1040.774,A -85,B 0,C 180,E1 32647.614,E2 32647.614} C_VEL
LIN {X 0,Y 699.059,Z 1021.655,A -85,B 0,C 180,E1 32646.122,E2 32646.122} C_VEL
LIN {X 0,Y 699.745,Z 1002.41,A -85,B 0,C 180,E1 32644.797,E2 32644.797} C_VEL
LIN {X 0,Y 700.495,Z 981.558,A -85,B 0,C 180,E1 32643.554,E2 32643.554} C_VEL
LIN {X 0,Y 701.196,Z 961.864,A -85,B 0,C 180,E1 32642.529,E2 32642.529} C_VEL
LIN {X 0,Y 701.931,Z 938.73,A -85,B 0,C 180,E1 32641.497,E2 32641.497} C_VEL
LIN {X 0,Y 702.56,Z 917.973,A -85,B 0,C 180,E1 32640.717,E2 32640.717} C_VEL
LIN {X 0,Y 703.223,Z 893.036,A -85,B 0,C 180,E1 32639.946,E2 32639.946} C_VEL
LIN {X 0,Y 703.674,Z 871.101,A -85,B 0,C 180,E1 32639.413,E2 32639.413} C_VEL
LIN {X 0,Y 704.193,Z 846.373,A -85,B 0,C 180,E1 32638.963,E2 32638.963} C_VEL
LIN {X 0,Y 704.531,Z 797.612,A -85,B 0,C 180,E1 32638.378,E2 32638.378} C_VEL
LIN {X 0,Y 705.903,Z 574.42,A -85,B 0,C 180,E1 32635.797,E2 32635.797} C_VEL
LIN {X 0,Y 706.535,Z 466.712,A -85,B 0,C 180,E1 32634.526,E2 32634.526} C_VEL
LIN {X 0,Y 703.195,Z 452.747,A -85,B 0,C 180,E1 32634.138,E2 32634.138} C_VEL
LIN {X 0,Y 703.836,Z 425.225,A -85,B 0,C 180,E1 32632.174,E2 32632.174} C_VEL
LIN {X 0,Y 696.376,Z 405.681,A -85,B 0,C 180,E1 32630.216,E2 32630.216} C_VEL
LIN {X 0,Y 696.402,Z 405.482,A -85,B 0,C 180,E1 32627.44,E2 32627.44} C_VEL
LIN {X 0,Y 696.36,Z 405.485,A -85,B 0,C 180,E1 32624.468,E2 32624.468} C_VEL
LIN {X 0,Y 696.401,Z 405.455,A -85,B 0,C 180,E1 32621.555,E2 32621.555} C_VEL
LIN {X 0,Y 696.372,Z 405.483,A -85,B 0,C 180,E1 32618.506,E2 32618.506} C_VEL
LIN {X 0,Y 696.398,Z 405.485,A -85,B 0,C 180,E1 32615.556,E2 32615.556} C_VEL
LIN {X 0,Y 696.382,Z 405.475,A -85,B 0,C 180,E1 32612.48,E2 32612.48} C_VEL
LIN {X 0,Y 696.402,Z 405.481,A -85,B 0,C 180,E1 32609.504,E2 32609.504} C_VEL
LIN {X 0,Y 696.388,Z 405.479,A -85,B 0,C 180,E1 32606.368,E2 32606.368} C_VEL
LIN {X 0,Y 696.399,Z 405.48,A -85,B 0,C 180,E1 32603.346,E2 32603.346} C_VEL
LIN {X 0,Y 696.397,Z 405.476,A -85,B 0,C 180,E1 32600.332,E2 32600.332} C_VEL
LIN {X 0,Y 696.398,Z 405.488,A -85,B 0,C 180,E1 32597.29,E2 32597.29} C_VEL
LIN {X 0,Y 696.397,Z 405.47,A -85,B 0,C 180,E1 32594.213,E2 32594.213} C_VEL
LIN {X 0,Y 696.392,Z 405.486,A -85,B 0,C 180,E1 32591.177,E2 32591.177} C_VEL
LIN {X 0,Y 696.4,Z 405.469,A -85,B 0,C 180,E1 32588.172,E2 32588.172} C_VEL
LIN {X 0,Y 696.388,Z 405.484,A -85,B 0,C 180,E1 32585.107,E2 32585.107} C_VEL
LIN {X 0,Y 696.398,Z 405.473,A -85,B 0,C 180,E1 32582.057,E2 32582.057} C_VEL
LIN {X 0,Y 696.382,Z 405.481,A -85,B 0,C 180,E1 32579.013,E2 32579.013} C_VEL
LIN {X 0,Y 696.39,Z 405.475,A -85,B 0,C 180,E1 32576.048,E2 32576.048} C_VEL
LIN {X 0,Y 696.373,Z 405.479,A -85,B 0,C 180,E1 32572.907,E2 32572.907} C_VEL
LIN {X 0,Y 696.379,Z 405.478,A -85,B 0,C 180,E1 32569.995,E2 32569.995} C_VEL
LIN {X 0,Y 696.373,Z 405.478,A -85,B 0,C 180,E1 32566.887,E2 32566.887} C_VEL
LIN {X 0,Y 696.357,Z 405.482,A -85,B 0,C 180,E1 32564.082,E2 32564.082} C_VEL
LIN {X 0,Y 696.395,Z 405.479,A -85,B 0,C 180,E1 32561.065,E2 32561.065} C_VEL
LIN {X 0,Y 696.339,Z 405.485,A -85,B 0,C 180,E1 32558.255,E2 32558.255} C_VEL
LIN {X 0,Y 696.403,Z 405.473,A -85,B 0,C 180,E1 32555.394,E2 32555.394} C_VEL
LIN {X 0,Y 696.404,Z 405.475,A -85,B 0,C 180,E1 32555.236,E2 32555.236} C_VEL
LIN {X 0,Y 695.408,Z 405.609,A -85,B 0,C 180,E1 32554.602,E2 32554.602} C_VEL
LIN {X 0,Y 688.944,Z 406.411,A -85,B 0,C 180,E1 32552.827,E2 32552.827} C_VEL
LIN {X 0,Y 688.396,Z 406.471,A -85,B 0,C 180,E1 32552.365,E2 32552.365} C_VEL
LIN {X 0,Y 688.41,Z 406.473,A -85,B 0,C 180,E1 32549.735,E2 32549.735} C_VEL
LIN {X 0,Y 688.41,Z 406.477,A -85,B 0,C 180,E1 32546.6,E2 32546.6} C_VEL
LIN {X 0,Y 688.381,Z 406.474,A -85,B 0,C 180,E1 32544.004,E2 32544.004} C_VEL
LIN {X 0,Y 688.463,Z 406.475,A -85,B 0,C 180,E1 32541.14,E2 32541.14} C_VEL
LIN {X 0,Y 688.379,Z 406.448,A -85,B 0,C 180,E1 32538.297,E2 32538.297} C_VEL
LIN {X 0,Y 688.372,Z 406.475,A -85,B 0,C 180,E1 32535.795,E2 32535.795} C_VEL
LIN {X 0,Y 688.45,Z 406.452,A -85,B 0,C 180,E1 32532.935,E2 32532.935} C_VEL
LIN {X 0,Y 688.362,Z 406.483,A -85,B 0,C 180,E1 32530.048,E2 32530.048} C_VEL
LIN {X 0,Y 688.356,Z 406.467,A -85,B 0,C 180,E1 32527.701,E2 32527.701} C_VEL
LIN {X 0,Y 688.446,Z 406.463,A -85,B 0,C 180,E1 32524.855,E2 32524.855} C_VEL
LIN {X 0,Y 688.44,Z 406.828,A -85,B 0,C 180,E1 32524.301,E2 32524.301} C_VEL
LIN {X 0,Y 691.094,Z 414.213,A -85,B 0,C 180,E1 32523.515,E2 32523.515} C_VEL
LIN {X 0,Y 700.169,Z 430.415,A -85,B 0,C 180,E1 32522.755,E2 32522.755} C_VEL
LIN {X 0,Y 698.267,Z 679.85,A -85,B 0,C 180,E1 32519.822,E2 32519.822} C_VEL
LIN {X 0,Y 697.341,Z 803.364,A -85,B 0,C 180,E1 32518.373,E2 32518.373} C_VEL
LIN {X 0,Y 696.842,Z 828.764,A -85,B 0,C 180,E1 32517.928,E2 32517.928} C_VEL
LIN {X 0,Y 696.281,Z 850.574,A -85,B 0,C 180,E1 32517.408,E2 32517.408} C_VEL
LIN {X 0,Y 695.588,Z 875.604,A -85,B 0,C 180,E1 32516.647,E2 32516.647} C_VEL
LIN {X 0,Y 694.899,Z 895.743,A -85,B 0,C 180,E1 32515.899,E2 32515.899} C_VEL
LIN {X 0,Y 694.089,Z 918.183,A -85,B 0,C 180,E1 32514.921,E2 32514.921} C_VEL
LIN {X 0,Y 693.248,Z 939.467,A -85,B 0,C 180,E1 32513.819,E2 32513.819} C_VEL
LIN {X 0,Y 692.434,Z 959.523,A -85,B 0,C 180,E1 32512.633,E2 32512.633} C_VEL
LIN {X 0,Y 691.593,Z 979.711,A -85,B 0,C 180,E1 32511.252,E2 32511.252} C_VEL
LIN {X 0,Y 690.848,Z 998.49,A -85,B 0,C 180,E1 32509.796,E2 32509.796} C_VEL
LIN {X 0,Y 690.152,Z 1015.977,A -85,B 0,C 180,E1 32508.237,E2 32508.237} C_VEL
LIN {X 0,Y 689.56,Z 1032.587,A -85,B 0,C 180,E1 32506.568,E2 32506.568} C_VEL
LIN {X 0,Y 689.093,Z 1047.13,A -85,B 0,C 180,E1 32504.882,E2 32504.882} C_VEL
LIN {X 0,Y 688.696,Z 1061.147,A -85,B 0,C 180,E1 32503.042,E2 32503.042} C_VEL
LIN {X 0,Y 688.387,Z 1072.965,A -85,B 0,C 180,E1 32501.224,E2 32501.224} C_VEL
LIN {X 0,Y 688.189,Z 1082.989,A -85,B 0,C 180,E1 32499.45,E2 32499.45} C_VEL
LIN {X 0,Y 688.059,Z 1092.495,A -85,B 0,C 180,E1 32497.431,E2 32497.431} C_VEL
LIN {X 0,Y 687.957,Z 1099.338,A -85,B 0,C 180,E1 32495.672,E2 32495.672} C_VEL
LIN {X 0,Y 687.912,Z 1105.778,A -85,B 0,C 180,E1 32493.583,E2 32493.583} C_VEL
LIN {X 0,Y 687.921,Z 1109.893,A -85,B 0,C 180,E1 32491.749,E2 32491.749} C_VEL
LIN {X 0,Y 687.909,Z 1112.96,A -85,B 0,C 180,E1 32489.75,E2 32489.75} C_VEL
LIN {X 0,Y 687.901,Z 1114.294,A -85,B 0,C 180,E1 32487.751,E2 32487.751} C_VEL
LIN {X 0,Y 687.906,Z 1114.251,A -85,B 0,C 180,E1 32485.999,E2 32485.999} C_VEL
LIN {X 0,Y 687.917,Z 1112.51,A -85,B 0,C 180,E1 32483.825,E2 32483.825} C_VEL
LIN {X 0,Y 687.921,Z 1109.549,A -85,B 0,C 180,E1 32481.979,E2 32481.979} C_VEL
LIN {X 0,Y 687.944,Z 1104.801,A -85,B 0,C 180,E1 32479.955,E2 32479.955} C_VEL
LIN {X 0,Y 687.96,Z 1098.804,A -85,B 0,C 180,E1 32478.089,E2 32478.089} C_VEL
LIN {X 0,Y 688.064,Z 1092.096,A -85,B 0,C 180,E1 32476.384,E2 32476.384} C_VEL
LIN {X 0,Y 688.21,Z 1082.241,A -85,B 0,C 180,E1 32474.322,E2 32474.322} C_VEL
LIN {X 0,Y 688.399,Z 1072.379,A -85,B 0,C 180,E1 32472.59,E2 32472.59} C_VEL
LIN {X 0,Y 688.717,Z 1059.704,A -85,B 0,C 180,E1 32470.67,E2 32470.67} C_VEL
LIN {X 0,Y 689.101,Z 1046.888,A -85,B 0,C 180,E1 32468.998,E2 32468.998} C_VEL
LIN {X 0,Y 689.603,Z 1031.463,A -85,B 0,C 180,E1 32467.223,E2 32467.223} C_VEL
LIN {X 0,Y 690.146,Z 1016.108,A -85,B 0,C 180,E1 32465.687,E2 32465.687} C_VEL
LIN {X 0,Y 690.853,Z 998.454,A -85,B 0,C 180,E1 32464.111,E2 32464.111} C_VEL
LIN {X 0,Y 691.583,Z 979.947,A -85,B 0,C 180,E1 32462.675,E2 32462.675} C_VEL
LIN {X 0,Y 692.419,Z 959.98,A -85,B 0,C 180,E1 32461.305,E2 32461.305} C_VEL
LIN {X 0,Y 693.242,Z 939.543,A -85,B 0,C 180,E1 32460.095,E2 32460.095} C_VEL
LIN {X 0,Y 694.114,Z 917.458,A -85,B 0,C 180,E1 32458.955,E2 32458.955} C_VEL
LIN {X 0,Y 694.886,Z 896.122,A -85,B 0,C 180,E1 32458.026,E2 32458.026} C_VEL
LIN {X 0,Y 695.622,Z 874.776,A -85,B 0,C 180,E1 32457.234,E2 32457.234} C_VEL
LIN {X 0,Y 696.296,Z 850.061,A -85,B 0,C 180,E1 32456.488,E2 32456.488} C_VEL
LIN {X 0,Y 696.867,Z 828.022,A -85,B 0,C 180,E1 32455.966,E2 32455.966} C_VEL
LIN {X 0,Y 697.346,Z 802.687,A -85,B 0,C 180,E1 32455.527,E2 32455.527} C_VEL
LIN {X 0,Y 699.211,Z 552.363,A -85,B 0,C 180,E1 32452.598,E2 32452.598} C_VEL
LIN {X 0,Y 700.001,Z 430.013,A -85,B 0,C 180,E1 32451.14,E2 32451.14} C_VEL
LIN {X 0,Y 691.08,Z 414.196,A -85,B 0,C 180,E1 32450.395,E2 32450.395} C_VEL
LIN {X 0,Y 688.41,Z 406.656,A -85,B 0,C 180,E1 32449.578,E2 32449.578} C_VEL
LIN {X 0,Y 688.379,Z 406.484,A -85,B 0,C 180,E1 32446.454,E2 32446.454} C_VEL
LIN {X 0,Y 688.367,Z 406.482,A -85,B 0,C 180,E1 32443.907,E2 32443.907} C_VEL
LIN {X 0,Y 688.458,Z 406.451,A -85,B 0,C 180,E1 32441.031,E2 32441.031} C_VEL
LIN {X 0,Y 688.381,Z 406.476,A -85,B 0,C 180,E1 32438.203,E2 32438.203} C_VEL
LIN {X 0,Y 688.378,Z 406.448,A -85,B 0,C 180,E1 32435.711,E2 32435.711} C_VEL
LIN {X 0,Y 688.466,Z 406.473,A -85,B 0,C 180,E1 32432.801,E2 32432.801} C_VEL
LIN {X 0,Y 688.389,Z 406.449,A -85,B 0,C 180,E1 32429.978,E2 32429.978} C_VEL
LIN {X 0,Y 688.404,Z 406.469,A -85,B 0,C 180,E1 32427.415,E2 32427.415} C_VEL
LIN {X 0,Y 688.438,Z 406.466,A -85,B 0,C 180,E1 32424.361,E2 32424.361} C_VEL
LIN {X 0,Y 688.399,Z 406.476,A -85,B 0,C 180,E1 32421.628,E2 32421.628} C_VEL
LIN {X 0,Y 688.467,Z 406.476,A -85,B 0,C 180,E1 32418.722,E2 32418.722} C_VEL
LIN {X 0,Y 688.409,Z 406.464,A -85,B 0,C 180,E1 32415.76,E2 32415.76} C_VEL
LIN {X 0,Y 688.453,Z 406.477,A -85,B 0,C 180,E1 32412.924,E2 32412.924} C_VEL
LIN {X 0,Y 688.427,Z 406.47,A -85,B 0,C 180,E1 32409.869,E2 32409.869} C_VEL
LIN {X 0,Y 688.438,Z 406.471,A -85,B 0,C 180,E1 32407.008,E2 32407.008} C_VEL
LIN {X 0,Y 688.439,Z 406.468,A -85,B 0,C 180,E1 32403.831,E2 32403.831} C_VEL
LIN {X 0,Y 688.455,Z 406.469,A -85,B 0,C 180,E1 32400.832,E2 32400.832} C_VEL
LIN {X 0,Y 688.445,Z 406.461,A -85,B 0,C 180,E1 32397.753,E2 32397.753} C_VEL
LIN {X 0,Y 688.459,Z 406.476,A -85,B 0,C 180,E1 32394.75,E2 32394.75} C_VEL
LIN {X 0,Y 688.451,Z 406.463,A -85,B 0,C 180,E1 32391.649,E2 32391.649} C_VEL
LIN {X 0,Y 688.459,Z 406.469,A -85,B 0,C 180,E1 32388.608,E2 32388.608} C_VEL
LIN {X 0,Y 688.456,Z 406.467,A -85,B 0,C 180,E1 32385.534,E2 32385.534} C_VEL
LIN {X 0,Y 688.459,Z 406.471,A -85,B 0,C 180,E1 32382.504,E2 32382.504} C_VEL
LIN {X 0,Y 688.458,Z 406.463,A -85,B 0,C 180,E1 32379.423,E2 32379.423} C_VEL
LIN {X 0,Y 688.453,Z 406.477,A -85,B 0,C 180,E1 32376.368,E2 32376.368} C_VEL
LIN {X 0,Y 688.459,Z 406.457,A -85,B 0,C 180,E1 32373.334,E2 32373.334} C_VEL
LIN {X 0,Y 688.447,Z 406.473,A -85,B 0,C 180,E1 32370.288,E2 32370.288} C_VEL
LIN {X 0,Y 688.464,Z 406.466,A -85,B 0,C 180,E1 32367.237,E2 32367.237} C_VEL
LIN {X 0,Y 688.437,Z 406.471,A -85,B 0,C 180,E1 32364.14,E2 32364.14} C_VEL
LIN {X 0,Y 688.468,Z 406.464,A -85,B 0,C 180,E1 32361.12,E2 32361.12} C_VEL
LIN {X 0,Y 688.43,Z 406.467,A -85,B 0,C 180,E1 32358.043,E2 32358.043} C_VEL
LIN {X 0,Y 688.453,Z 406.47,A -85,B 0,C 180,E1 32355.101,E2 32355.101} C_VEL
LIN {X 0,Y 688.428,Z 406.468,A -85,B 0,C 180,E1 32352.034,E2 32352.034} C_VEL
LIN {X 0,Y 688.476,Z 406.682,A -85,B 0,C 180,E1 32350.221,E2 32350.221} C_VEL
LIN {X 0,Y 696.889,Z 429.079,A -85,B 0,C 180,E1 32347.962,E2 32347.962} C_VEL
LIN {X 0,Y 696.264,Z 452.957,A -85,B 0,C 180,E1 32346.265,E2 32346.265} C_VEL
LIN {X 0,Y 700.161,Z 469.991,A -85,B 0,C 180,E1 32345.806,E2 32345.806} C_VEL
LIN {X 0,Y 698.274,Z 717.706,A -85,B 0,C 180,E1 32342.893,E2 32342.893} C_VEL
LIN {X 0,Y 697.352,Z 843.23,A -85,B 0,C 180,E1 32341.42,E2 32341.42} C_VEL
LIN {X 0,Y 696.839,Z 868.75,A -85,B 0,C 180,E1 32340.973,E2 32340.973} C_VEL
LIN {X 0,Y 696.274,Z 890.553,A -85,B 0,C 180,E1 32340.454,E2 32340.454} C_VEL
LIN {X 0,Y 695.634,Z 914.552,A -85,B 0,C 180,E1 32339.729,E2 32339.729} C_VEL
LIN {X 0,Y 694.916,Z 935.348,A -85,B 0,C 180,E1 32338.959,E2 32338.959} C_VEL
LIN {X 0,Y 694.117,Z 957.248,A -85,B 0,C 180,E1 32338.009,E2 32338.009} C_VEL
LIN {X 0,Y 693.26,Z 979.134,A -85,B 0,C 180,E1 32336.883,E2 32336.883} C_VEL
LIN {X 0,Y 692.486,Z 998.176,A -85,B 0,C 180,E1 32335.761,E2 32335.761} C_VEL
LIN {X 0,Y 691.612,Z 1019.228,A -85,B 0,C 180,E1 32334.333,E2 32334.333} C_VEL
LIN {X 0,Y 690.896,Z 1037.054,A -85,B 0,C 180,E1 32332.957,E2 32332.957} C_VEL
LIN {X 0,Y 690.213,Z 1054.604,A -85,B 0,C 180,E1 32331.412,E2 32331.412} C_VEL
LIN {X 0,Y 689.67,Z 1069.637,A -85,B 0,C 180,E1 32329.92,E2 32329.92} C_VEL
LIN {X 0,Y 689.134,Z 1085.812,A -85,B 0,C 180,E1 32328.09,E2 32328.09} C_VEL
LIN {X 0,Y 688.752,Z 1098.528,A -85,B 0,C 180,E1 32326.445,E2 32326.445} C_VEL
LIN {X 0,Y 688.429,Z 1111.76,A -85,B 0,C 180,E1 32324.467,E2 32324.467} C_VEL
LIN {X 0,Y 688.231,Z 1121.568,A -85,B 0,C 180,E1 32322.758,E2 32322.758} C_VEL
LIN {X 0,Y 688.062,Z 1131.475,A -85,B 0,C 180,E1 32320.72,E2 32320.72} C_VEL
LIN {X 0,Y 687.969,Z 1138.513,A -85,B 0,C 180,E1 32318.947,E2 32318.947} C_VEL
LIN {X 0,Y 687.931,Z 1144.252,A -85,B 0,C 180,E1 32317.181,E2 32317.181} C_VEL
LIN {X 0,Y 687.891,Z 1149.338,A -85,B 0,C 180,E1 32315.087,E2 32315.087} C_VEL
LIN {X 0,Y 687.903,Z 1152.236,A -85,B 0,C 180,E1 32313.333,E2 32313.333} C_VEL
LIN {X 0,Y 687.909,Z 1154.171,A -85,B 0,C 180,E1 32311.249,E2 32311.249} C_VEL
LIN {X 0,Y 687.882,Z 1154.351,A -85,B 0,C 180,E1 32309.417,E2 32309.417} C_VEL
LIN {X 0,Y 687.905,Z 1153.296,A -85,B 0,C 180,E1 32307.584,E2 32307.584} C_VEL
LIN {X 0,Y 687.919,Z 1150.449,A -85,B 0,C 180,E1 32305.498,E2 32305.498} C_VEL
LIN {X 0,Y 687.929,Z 1146.689,A -85,B 0,C 180,E1 32303.742,E2 32303.742} C_VEL
LIN {X 0,Y 687.977,Z 1141.141,A -85,B 0,C 180,E1 32301.792,E2 32301.792} C_VEL
LIN {X 0,Y 688.037,Z 1133.604,A -85,B 0,C 180,E1 32299.788,E2 32299.788} C_VEL
LIN {X 0,Y 688.156,Z 1125.524,A -85,B 0,C 180,E1 32298.008,E2 32298.008} C_VEL
LIN {X 0,Y 688.37,Z 1114.356,A -85,B 0,C 180,E1 32295.961,E2 32295.961} C_VEL
LIN {X 0,Y 688.624,Z 1103.384,A -85,B 0,C 180,E1 32294.245,E2 32294.245} C_VEL
LIN {X 0,Y 689.012,Z 1089.332,A -85,B 0,C 180,E1 32292.344,E2 32292.344} C_VEL
LIN {X 0,Y 689.473,Z 1075.299,A -85,B 0,C 180,E1 32290.692,E2 32290.692} C_VEL
LIN {X 0,Y 690.082,Z 1058.176,A -85,B 0,C 180,E1 32288.927,E2 32288.927} C_VEL
LIN {X 0,Y 690.7,Z 1041.787,A -85,B 0,C 180,E1 32287.441,E2 32287.441} C_VEL
LIN {X 0,Y 691.498,Z 1022.26,A -85,B 0,C 180,E1 32285.89,E2 32285.89} C_VEL
LIN {X 0,Y 692.24,Z 1003.742,A -85,B 0,C 180,E1 32284.596,E2 32284.596} C_VEL
LIN {X 0,Y 693.127,Z 982.363,A -85,B 0,C 180,E1 32283.297,E2 32283.297} C_VEL
LIN {X 0,Y 693.907,Z 962.761,A -85,B 0,C 180,E1 32282.262,E2 32282.262} C_VEL
LIN {X 0,Y 694.792,Z 938.734,A -85,B 0,C 180,E1 32281.177,E2 32281.177} C_VEL
LIN {X 0,Y 695.505,Z 917.827,A -85,B 0,C 180,E1 32280.386,E2 32280.386} C_VEL
LIN {X 0,Y 696.237,Z 892.931,A -85,B 0,C 180,E1 32279.61,E2 32279.61} C_VEL
LIN {X 0,Y 696.764,Z 870.969,A -85,B 0,C 180,E1 32279.074,E2 32279.074} C_VEL
LIN {X 0,Y 697.33,Z 846.159,A -85,B 0,C 180,E1 32278.621,E2 32278.621} C_VEL
LIN {X 0,Y 697.731,Z 795.407,A -85,B 0,C 180,E1 32278.007,E2 32278.007} C_VEL
LIN {X 0,Y 699.289,Z 573.503,A -85,B 0,C 180,E1 32275.417,E2 32275.417} C_VEL
LIN {X 0,Y 699.974,Z 468.396,A -85,B 0,C 180,E1 32274.163,E2 32274.163} C_VEL
LIN {X 0,Y 696.249,Z 452.736,A -85,B 0,C 180,E1 32273.724,E2 32273.724} C_VEL
LIN {X 0,Y 696.746,Z 428.515,A -85,B 0,C 180,E1 32271.987,E2 32271.987} C_VEL
LIN {X 0,Y 688.476,Z 406.671,A -85,B 0,C 180,E1 32269.77,E2 32269.77} C_VEL
LIN {X 0,Y 688.429,Z 406.476,A -85,B 0,C 180,E1 32266.691,E2 32266.691} C_VEL
LIN {X 0,Y 688.444,Z 406.476,A -85,B 0,C 180,E1 32263.793,E2 32263.793} C_VEL
LIN {X 0,Y 688.442,Z 406.454,A -85,B 0,C 180,E1 32260.698,E2 32260.698} C_VEL
LIN {X 0,Y 688.451,Z 406.476,A -85,B 0,C 180,E1 32257.695,E2 32257.695} C_VEL
LIN {X 0,Y 688.448,Z 406.47,A -85,B 0,C 180,E1 32254.563,E2 32254.563} C_VEL
LIN {X 0,Y 688.46,Z 406.474,A -85,B 0,C 180,E1 32251.511,E2 32251.511} C_VEL
LIN {X 0,Y 688.451,Z 406.459,A -85,B 0,C 180,E1 32248.449,E2 32248.449} C_VEL
LIN {X 0,Y 688.46,Z 406.47,A -85,B 0,C 180,E1 32245.395,E2 32245.395} C_VEL
LIN {X 0,Y 688.449,Z 406.467,A -85,B 0,C 180,E1 32242.276,E2 32242.276} C_VEL
LIN {X 0,Y 688.455,Z 406.467,A -85,B 0,C 180,E1 32239.25,E2 32239.25} C_VEL
LIN {X 0,Y 688.456,Z 406.467,A -85,B 0,C 180,E1 32236.192,E2 32236.192} C_VEL
LIN {X 0,Y 688.454,Z 406.471,A -85,B 0,C 180,E1 32233.181,E2 32233.181} C_VEL
LIN {X 0,Y 688.46,Z 406.465,A -85,B 0,C 180,E1 32230.121,E2 32230.121} C_VEL
LIN {X 0,Y 688.448,Z 406.476,A -85,B 0,C 180,E1 32227.091,E2 32227.091} C_VEL
LIN {X 0,Y 688.461,Z 406.462,A -85,B 0,C 180,E1 32224.081,E2 32224.081} C_VEL
LIN {X 0,Y 688.442,Z 406.476,A -85,B 0,C 180,E1 32220.999,E2 32220.999} C_VEL
LIN {X 0,Y 688.457,Z 406.461,A -85,B 0,C 180,E1 32218.002,E2 32218.002} C_VEL
LIN {X 0,Y 688.436,Z 406.476,A -85,B 0,C 180,E1 32214.917,E2 32214.917} C_VEL
LIN {X 0,Y 688.446,Z 406.459,A -85,B 0,C 180,E1 32211.985,E2 32211.985} C_VEL
LIN {X 0,Y 688.433,Z 406.475,A -85,B 0,C 180,E1 32208.862,E2 32208.862} C_VEL
LIN {X 0,Y 688.422,Z 406.461,A -85,B 0,C 180,E1 32206.048,E2 32206.048} C_VEL
LIN {X 0,Y 688.443,Z 406.474,A -85,B 0,C 180,E1 32202.939,E2 32202.939} C_VEL
LIN {X 0,Y 688.407,Z 406.468,A -85,B 0,C 180,E1 32200.13,E2 32200.13} C_VEL
LIN {X 0,Y 688.468,Z 406.471,A -85,B 0,C 180,E1 32197.184,E2 32197.184} C_VEL
LIN {X 0,Y 688.398,Z 406.475,A -85,B 0,C 180,E1 32194.352,E2 32194.352} C_VEL
LIN {X 0,Y 688.396,Z 406.471,A -85,B 0,C 180,E1 32192.365,E2 32192.365} C_VEL
LIN {X 0,Y 687.383,Z 406.597,A -85,B 0,C 180,E1 32191.724,E2 32191.724} C_VEL
LIN {X 0,Y 680.98,Z 407.398,A -85,B 0,C 180,E1 32189.927,E2 32189.927} C_VEL
LIN {X 0,Y 680.504,Z 407.461,A -85,B 0,C 180,E1 32189.46,E2 32189.46} C_VEL
LIN {X 0,Y 680.458,Z 407.465,A -85,B 0,C 180,E1 32186.426,E2 32186.426} C_VEL
LIN {X 0,Y 680.446,Z 407.463,A -85,B 0,C 180,E1 32183.896,E2 32183.896} C_VEL
LIN {X 0,Y 680.522,Z 407.464,A -85,B 0,C 180,E1 32180.925,E2 32180.925} C_VEL
LIN {X 0,Y 680.433,Z 407.433,A -85,B 0,C 180,E1 32178.152,E2 32178.152} C_VEL
LIN {X 0,Y 680.445,Z 407.464,A -85,B 0,C 180,E1 32175.575,E2 32175.575} C_VEL
LIN {X 0,Y 680.454,Z 407.435,A -85,B 0,C 180,E1 32172.467,E2 32172.467} C_VEL
LIN {X 0,Y 680.42,Z 407.472,A -85,B 0,C 180,E1 32169.845,E2 32169.845} C_VEL
LIN {X 0,Y 680.44,Z 407.453,A -85,B 0,C 180,E1 32167.346,E2 32167.346} C_VEL
LIN {X 0,Y 680.537,Z 407.641,A -85,B 0,C 180,E1 32164.782,E2 32164.782} C_VEL
LIN {X 0,Y 682.903,Z 414.404,A -85,B 0,C 180,E1 32164.032,E2 32164.032} C_VEL
LIN {X 0,Y 693.537,Z 433.026,A -85,B 0,C 180,E1 32163.12,E2 32163.12} C_VEL
LIN {X 0,Y 691.921,Z 635.391,A -85,B 0,C 180,E1 32160.705,E2 32160.705} C_VEL
LIN {X 0,Y 690.506,Z 803.186,A -85,B 0,C 180,E1 32158.723,E2 32158.723} C_VEL
LIN {X 0,Y 689.97,Z 828.501,A -85,B 0,C 180,E1 32158.277,E2 32158.277} C_VEL
LIN {X 0,Y 689.344,Z 850.256,A -85,B 0,C 180,E1 32157.757,E2 32157.757} C_VEL
LIN {X 0,Y 688.617,Z 874.164,A -85,B 0,C 180,E1 32157.032,E2 32157.032} C_VEL
LIN {X 0,Y 687.798,Z 895.481,A -85,B 0,C 180,E1 32156.237,E2 32156.237} C_VEL
LIN {X 0,Y 686.931,Z 917.004,A -85,B 0,C 180,E1 32155.296,E2 32155.296} C_VEL
LIN {X 0,Y 685.946,Z 939.18,A -85,B 0,C 180,E1 32154.145,E2 32154.145} C_VEL
LIN {X 0,Y 685.036,Z 959.437,A -85,B 0,C 180,E1 32152.937,E2 32152.937} C_VEL
LIN {X 0,Y 684.066,Z 979.89,A -85,B 0,C 180,E1 32151.524,E2 32151.524} C_VEL
LIN {X 0,Y 683.225,Z 999.019,A -85,B 0,C 180,E1 32150.022,E2 32150.022} C_VEL
LIN {X 0,Y 682.442,Z 1016.376,A -85,B 0,C 180,E1 32148.45,E2 32148.45} C_VEL
LIN {X 0,Y 681.796,Z 1032.655,A -85,B 0,C 180,E1 32146.793,E2 32146.793} C_VEL
LIN {X 0,Y 681.244,Z 1047.637,A -85,B 0,C 180,E1 32145.032,E2 32145.032} C_VEL
LIN {X 0,Y 680.782,Z 1061.708,A -85,B 0,C 180,E1 32143.15,E2 32143.15} C_VEL
LIN {X 0,Y 680.452,Z 1073.19,A -85,B 0,C 180,E1 32141.356,E2 32141.356} C_VEL
LIN {X 0,Y 680.221,Z 1083.64,A -85,B 0,C 180,E1 32139.476,E2 32139.476} C_VEL
LIN {X 0,Y 680.079,Z 1092.648,A -85,B 0,C 180,E1 32137.519,E2 32137.519} C_VEL
LIN {X 0,Y 679.967,Z 1099.468,A -85,B 0,C 180,E1 32135.739,E2 32135.739} C_VEL
LIN {X 0,Y 679.918,Z 1105.865,A -85,B 0,C 180,E1 32133.626,E2 32133.626} C_VEL
LIN {X 0,Y 679.922,Z 1109.803,A -85,B 0,C 180,E1 32131.854,E2 32131.854} C_VEL
LIN {X 0,Y 679.92,Z 1112.783,A -85,B 0,C 180,E1 32129.916,E2 32129.916} C_VEL
LIN {X 0,Y 679.904,Z 1114.281,A -85,B 0,C 180,E1 32127.809,E2 32127.809} C_VEL
LIN {X 0,Y 679.904,Z 1114.263,A -85,B 0,C 180,E1 32126.037,E2 32126.037} C_VEL
LIN {X 0,Y 679.917,Z 1112.575,A -85,B 0,C 180,E1 32123.837,E2 32123.837} C_VEL
LIN {X 0,Y 679.923,Z 1109.641,A -85,B 0,C 180,E1 32121.969,E2 32121.969} C_VEL
LIN {X 0,Y 679.948,Z 1104.948,A -85,B 0,C 180,E1 32119.922,E2 32119.922} C_VEL
LIN {X 0,Y 679.979,Z 1098.672,A -85,B 0,C 180,E1 32117.947,E2 32117.947} C_VEL
LIN {X 0,Y 680.086,Z 1091.583,A -85,B 0,C 180,E1 32116.134,E2 32116.134} C_VEL
LIN {X 0,Y 680.277,Z 1081.574,A -85,B 0,C 180,E1 32114.046,E2 32114.046} C_VEL
LIN {X 0,Y 680.496,Z 1071.624,A -85,B 0,C 180,E1 32112.292,E2 32112.292} C_VEL
LIN {X 0,Y 680.882,Z 1058.127,A -85,B 0,C 180,E1 32110.259,E2 32110.259} C_VEL
LIN {X 0,Y 681.315,Z 1045.134,A -85,B 0,C 180,E1 32108.566,E2 32108.566} C_VEL
LIN {X 0,Y 681.963,Z 1028.494,A -85,B 0,C 180,E1 32106.679,E2 32106.679} C_VEL
LIN {X 0,Y 682.587,Z 1013.025,A -85,B 0,C 180,E1 32105.139,E2 32105.139} C_VEL
LIN {X 0,Y 683.426,Z 994.211,A -85,B 0,C 180,E1 32103.498,E2 32103.498} C_VEL
LIN {X 0,Y 684.23,Z 976.281,A -85,B 0,C 180,E1 32102.119,E2 32102.119} C_VEL
LIN {X 0,Y 685.203,Z 955.61,A -85,B 0,C 180,E1 32100.735,E2 32100.735} C_VEL
LIN {X 0,Y 686.089,Z 935.748,A -85,B 0,C 180,E1 32099.573,E2 32099.573} C_VEL
LIN {X 0,Y 687.123,Z 912.491,A -85,B 0,C 180,E1 32098.408,E2 32098.408} C_VEL
LIN {X 0,Y 687.901,Z 892.781,A -85,B 0,C 180,E1 32097.564,E2 32097.564} C_VEL
LIN {X 0,Y 688.785,Z 868.601,A -85,B 0,C 180,E1 32096.695,E2 32096.695} C_VEL
LIN {X 0,Y 689.465,Z 846.853,A -85,B 0,C 180,E1 32096.065,E2 32096.065} C_VEL
LIN {X 0,Y 690.147,Z 822.444,A -85,B 0,C 180,E1 32095.509,E2 32095.509} C_VEL
LIN {X 0,Y 690.539,Z 799.099,A -85,B 0,C 180,E1 32095.131,E2 32095.131} C_VEL
LIN {X 0,Y 692.619,Z 550.483,A -85,B 0,C 180,E1 32092.201,E2 32092.201} C_VEL
LIN {X 0,Y 693.496,Z 432.949,A -85,B 0,C 180,E1 32090.787,E2 32090.787} C_VEL
LIN {X 0,Y 684.236,Z 416.873,A -85,B 0,C 180,E1 32090.005,E2 32090.005} C_VEL
LIN {X 0,Y 682.792,Z 414.099,A -85,B 0,C 180,E1 32089.856,E2 32089.856} C_VEL
LIN {X 0,Y 680.533,Z 407.637,A -85,B 0,C 180,E1 32089.125,E2 32089.125} C_VEL
LIN {X 0,Y 680.426,Z 407.474,A -85,B 0,C 180,E1 32086.2,E2 32086.2} C_VEL
LIN {X 0,Y 680.44,Z 407.472,A -85,B 0,C 180,E1 32083.682,E2 32083.682} C_VEL
LIN {X 0,Y 680.474,Z 407.452,A -85,B 0,C 180,E1 32080.613,E2 32080.613} C_VEL
LIN {X 0,Y 680.438,Z 407.465,A -85,B 0,C 180,E1 32078.004,E2 32078.004} C_VEL
LIN {X 0,Y 680.467,Z 407.437,A -85,B 0,C 180,E1 32075.36,E2 32075.36} C_VEL
LIN {X 0,Y 680.46,Z 407.462,A -85,B 0,C 180,E1 32072.236,E2 32072.236} C_VEL
LIN {X 0,Y 680.448,Z 407.435,A -85,B 0,C 180,E1 32069.684,E2 32069.684} C_VEL
LIN {X 0,Y 680.528,Z 407.462,A -85,B 0,C 180,E1 32066.813,E2 32066.813} C_VEL
LIN {X 0,Y 680.458,Z 407.457,A -85,B 0,C 180,E1 32063.835,E2 32063.835} C_VEL
LIN {X 0,Y 680.485,Z 407.467,A -85,B 0,C 180,E1 32061.19,E2 32061.19} C_VEL
LIN {X 0,Y 680.486,Z 407.461,A -85,B 0,C 180,E1 32058.062,E2 32058.062} C_VEL
LIN {X 0,Y 680.479,Z 407.456,A -85,B 0,C 180,E1 32055.25,E2 32055.25} C_VEL
LIN {X 0,Y 680.507,Z 407.452,A -85,B 0,C 180,E1 32052.129,E2 32052.129} C_VEL
LIN {X 0,Y 680.485,Z 407.464,A -85,B 0,C 180,E1 32049.216,E2 32049.216} C_VEL
LIN {X 0,Y 680.524,Z 407.453,A -85,B 0,C 180,E1 32046.157,E2 32046.157} C_VEL
LIN {X 0,Y 680.488,Z 407.463,A -85,B 0,C 180,E1 32043.201,E2 32043.201} C_VEL
LIN {X 0,Y 680.523,Z 407.457,A -85,B 0,C 180,E1 32040.168,E2 32040.168} C_VEL
LIN {X 0,Y 680.489,Z 407.454,A -85,B 0,C 180,E1 32037.221,E2 32037.221} C_VEL
LIN {X 0,Y 680.515,Z 407.457,A -85,B 0,C 180,E1 32034.266,E2 32034.266} C_VEL
LIN {X 0,Y 680.496,Z 407.455,A -85,B 0,C 180,E1 32031.295,E2 32031.295} C_VEL
LIN {X 0,Y 680.514,Z 407.453,A -85,B 0,C 180,E1 32028.387,E2 32028.387} C_VEL
LIN {X 0,Y 680.506,Z 407.459,A -85,B 0,C 180,E1 32025.361,E2 32025.361} C_VEL
LIN {X 0,Y 680.515,Z 407.462,A -85,B 0,C 180,E1 32022.381,E2 32022.381} C_VEL
LIN {X 0,Y 680.516,Z 407.453,A -85,B 0,C 180,E1 32019.351,E2 32019.351} C_VEL
LIN {X 0,Y 680.513,Z 407.466,A -85,B 0,C 180,E1 32016.351,E2 32016.351} C_VEL
LIN {X 0,Y 680.52,Z 407.446,A -85,B 0,C 180,E1 32013.281,E2 32013.281} C_VEL
LIN {X 0,Y 680.504,Z 407.46,A -85,B 0,C 180,E1 32010.222,E2 32010.222} C_VEL
LIN {X 0,Y 680.523,Z 407.456,A -85,B 0,C 180,E1 32007.168,E2 32007.168} C_VEL
LIN {X 0,Y 680.496,Z 407.459,A -85,B 0,C 180,E1 32004.107,E2 32004.107} C_VEL
LIN {X 0,Y 680.528,Z 407.453,A -85,B 0,C 180,E1 32001.142,E2 32001.142} C_VEL
LIN {X 0,Y 680.49,Z 407.455,A -85,B 0,C 180,E1 31998.031,E2 31998.031} C_VEL
LIN {X 0,Y 680.516,Z 407.457,A -85,B 0,C 180,E1 31995.09,E2 31995.09} C_VEL
LIN {X 0,Y 680.483,Z 407.457,A -85,B 0,C 180,E1 31991.969,E2 31991.969} C_VEL
LIN {X 0,Y 680.568,Z 407.756,A -85,B 0,C 180,E1 31990.667,E2 31990.667} C_VEL
LIN {X 0,Y 689.854,Z 432.253,A -85,B 0,C 180,E1 31988.157,E2 31988.157} C_VEL
LIN {X 0,Y 689.326,Z 453.096,A -85,B 0,C 180,E1 31986.672,E2 31986.672} C_VEL
LIN {X 0,Y 693.646,Z 471.844,A -85,B 0,C 180,E1 31986.171,E2 31986.171} C_VEL
LIN {X 0,Y 691.544,Z 718.978,A -85,B 0,C 180,E1 31983.239,E2 31983.239} C_VEL
LIN {X 0,Y 690.515,Z 843.293,A -85,B 0,C 180,E1 31981.766,E2 31981.766} C_VEL
LIN {X 0,Y 689.958,Z 868.748,A -85,B 0,C 180,E1 31981.317,E2 31981.317} C_VEL
LIN {X 0,Y 689.331,Z 890.442,A -85,B 0,C 180,E1 31980.797,E2 31980.797} C_VEL
LIN {X 0,Y 688.603,Z 914.548,A -85,B 0,C 180,E1 31980.064,E2 31980.064} C_VEL
LIN {X 0,Y 687.798,Z 935.574,A -85,B 0,C 180,E1 31979.278,E2 31979.278} C_VEL
LIN {X 0,Y 686.92,Z 957.252,A -85,B 0,C 180,E1 31978.329,E2 31978.329} C_VEL
LIN {X 0,Y 685.951,Z 979.049,A -85,B 0,C 180,E1 31977.197,E2 31977.197} C_VEL
LIN {X 0,Y 685.058,Z 998.953,A -85,B 0,C 180,E1 31976.012,E2 31976.012} C_VEL
LIN {X 0,Y 684.091,Z 1019.29,A -85,B 0,C 180,E1 31974.613,E2 31974.613} C_VEL
LIN {X 0,Y 683.28,Z 1037.607,A -85,B 0,C 180,E1 31973.182,E2 31973.182} C_VEL
LIN {X 0,Y 682.486,Z 1055.533,A -85,B 0,C 180,E1 31971.576,E2 31971.576} C_VEL
LIN {X 0,Y 681.843,Z 1071.622,A -85,B 0,C 180,E1 31969.948,E2 31969.948} C_VEL
LIN {X 0,Y 681.255,Z 1087.228,A -85,B 0,C 180,E1 31968.129,E2 31968.129} C_VEL
LIN {X 0,Y 680.806,Z 1101.06,A -85,B 0,C 180,E1 31966.291,E2 31966.291} C_VEL
LIN {X 0,Y 680.463,Z 1113.321,A -85,B 0,C 180,E1 31964.379,E2 31964.379} C_VEL
LIN {X 0,Y 680.235,Z 1123.861,A -85,B 0,C 180,E1 31962.479,E2 31962.479} C_VEL
LIN {X 0,Y 680.076,Z 1132.896,A -85,B 0,C 180,E1 31960.505,E2 31960.505} C_VEL
LIN {X 0,Y 679.967,Z 1139.726,A -85,B 0,C 180,E1 31958.712,E2 31958.712} C_VEL
LIN {X 0,Y 679.928,Z 1146.07,A -85,B 0,C 180,E1 31956.587,E2 31956.587} C_VEL
LIN {X 0,Y 679.905,Z 1149.974,A -85,B 0,C 180,E1 31954.809,E2 31954.809} C_VEL
LIN {X 0,Y 679.883,Z 1152.911,A -85,B 0,C 180,E1 31952.866,E2 31952.866} C_VEL
LIN {X 0,Y 679.889,Z 1154.284,A -85,B 0,C 180,E1 31950.843,E2 31950.843} C_VEL
LIN {X 0,Y 679.889,Z 1154.284,A -85,B 0,C 180,E1 31949.157,E2 31949.157} C_VEL
LIN {X 0,Y 679.883,Z 1152.911,A -85,B 0,C 180,E1 31947.134,E2 31947.134} C_VEL
LIN {X 0,Y 679.905,Z 1149.973,A -85,B 0,C 180,E1 31945.191,E2 31945.191} C_VEL
LIN {X 0,Y 679.931,Z 1145.864,A -85,B 0,C 180,E1 31943.329,E2 31943.329} C_VEL
LIN {X 0,Y 679.969,Z 1139.423,A -85,B 0,C 180,E1 31941.203,E2 31941.203} C_VEL
LIN {X 0,Y 680.076,Z 1132.895,A -85,B 0,C 180,E1 31939.495,E2 31939.495} C_VEL
LIN {X 0,Y 680.235,Z 1123.862,A -85,B 0,C 180,E1 31937.521,E2 31937.521} C_VEL
LIN {X 0,Y 680.463,Z 1113.324,A -85,B 0,C 180,E1 31935.621,E2 31935.621} C_VEL
LIN {X 0,Y 680.806,Z 1101.063,A -85,B 0,C 180,E1 31933.709,E2 31933.709} C_VEL
LIN {X 0,Y 681.255,Z 1087.228,A -85,B 0,C 180,E1 31931.871,E2 31931.871} C_VEL
LIN {X 0,Y 681.843,Z 1071.621,A -85,B 0,C 180,E1 31930.052,E2 31930.052} C_VEL
LIN {X 0,Y 682.486,Z 1055.533,A -85,B 0,C 180,E1 31928.424,E2 31928.424} C_VEL
LIN {X 0,Y 683.28,Z 1037.607,A -85,B 0,C 180,E1 31926.818,E2 31926.818} C_VEL
LIN {X 0,Y 684.093,Z 1019.223,A -85,B 0,C 180,E1 31925.382,E2 31925.382} C_VEL
LIN {X 0,Y 685.089,Z 998.174,A -85,B 0,C 180,E1 31923.94,E2 31923.94} C_VEL
LIN {X 0,Y 685.95,Z 979.044,A -85,B 0,C 180,E1 31922.803,E2 31922.803} C_VEL
LIN {X 0,Y 686.92,Z 957.255,A -85,B 0,C 180,E1 31921.671,E2 31921.671} C_VEL
LIN {X 0,Y 687.798,Z 935.575,A -85,B 0,C 180,E1 31920.722,E2 31920.722} C_VEL
LIN {X 0,Y 688.61,Z 914.393,A -85,B 0,C 180,E1 31919.931,E2 31919.931} C_VEL
LIN {X 0,Y 689.341,Z 890.141,A -85,B 0,C 180,E1 31919.195,E2 31919.195} C_VEL
LIN {X 0,Y 689.972,Z 868.361,A -85,B 0,C 180,E1 31918.675,E2 31918.675} C_VEL
LIN {X 0,Y 690.517,Z 842.987,A -85,B 0,C 180,E1 31918.23,E2 31918.23} C_VEL
LIN {X 0,Y 692.528,Z 596.062,A -85,B 0,C 180,E1 31915.31,E2 31915.31} C_VEL
LIN {X 0,Y 693.498,Z 470.299,A -85,B 0,C 180,E1 31913.801,E2 31913.801} C_VEL
LIN {X 0,Y 689.27,Z 452.444,A -85,B 0,C 180,E1 31913.297,E2 31913.297} C_VEL
LIN {X 0,Y 689.861,Z 432.26,A -85,B 0,C 180,E1 31911.842,E2 31911.842} C_VEL
LIN {X 0,Y 681.411,Z 410.25,A -85,B 0,C 180,E1 31909.603,E2 31909.603} C_VEL
LIN {X 0,Y 680.546,Z 407.598,A -85,B 0,C 180,E1 31909.281,E2 31909.281} C_VEL
LIN {X 0,Y 680.478,Z 407.468,A -85,B 0,C 180,E1 31906.321,E2 31906.321} C_VEL
LIN {X 0,Y 680.523,Z 407.452,A -85,B 0,C 180,E1 31903.443,E2 31903.443} C_VEL
LIN {X 0,Y 680.485,Z 407.444,A -85,B 0,C 180,E1 31900.435,E2 31900.435} C_VEL
LIN {X 0,Y 680.523,Z 407.458,A -85,B 0,C 180,E1 31897.493,E2 31897.493} C_VEL
LIN {X 0,Y 680.5,Z 407.461,A -85,B 0,C 180,E1 31894.451,E2 31894.451} C_VEL
LIN {X 0,Y 680.523,Z 407.464,A -85,B 0,C 180,E1 31891.44,E2 31891.44} C_VEL
LIN {X 0,Y 680.505,Z 407.449,A -85,B 0,C 180,E1 31888.333,E2 31888.333} C_VEL
LIN {X 0,Y 680.518,Z 407.457,A -85,B 0,C 180,E1 31885.313,E2 31885.313} C_VEL
LIN {X 0,Y 680.507,Z 407.457,A -85,B 0,C 180,E1 31882.228,E2 31882.228} C_VEL
LIN {X 0,Y 680.514,Z 407.455,A -85,B 0,C 180,E1 31879.216,E2 31879.216} C_VEL
LIN {X 0,Y 680.519,Z 407.456,A -85,B 0,C 180,E1 31876.211,E2 31876.211} C_VEL
LIN {X 0,Y 680.514,Z 407.459,A -85,B 0,C 180,E1 31873.164,E2 31873.164} C_VEL
LIN {X 0,Y 680.519,Z 407.455,A -85,B 0,C 180,E1 31870.07,E2 31870.07} C_VEL
LIN {X 0,Y 680.503,Z 407.464,A -85,B 0,C 180,E1 31867.005,E2 31867.005} C_VEL
LIN {X 0,Y 680.52,Z 407.452,A -85,B 0,C 180,E1 31863.96,E2 31863.96} C_VEL
LIN {X 0,Y 680.497,Z 407.464,A -85,B 0,C 180,E1 31860.926,E2 31860.926} C_VEL
LIN {X 0,Y 680.519,Z 407.449,A -85,B 0,C 180,E1 31857.979,E2 31857.979} C_VEL
LIN {X 0,Y 680.493,Z 407.464,A -85,B 0,C 180,E1 31854.858,E2 31854.858} C_VEL
LIN {X 0,Y 680.517,Z 407.446,A -85,B 0,C 180,E1 31851.891,E2 31851.891} C_VEL
LIN {X 0,Y 680.49,Z 407.464,A -85,B 0,C 180,E1 31848.816,E2 31848.816} C_VEL
LIN {X 0,Y 680.49,Z 407.448,A -85,B 0,C 180,E1 31845.969,E2 31845.969} C_VEL
LIN {X 0,Y 680.49,Z 407.462,A -85,B 0,C 180,E1 31842.822,E2 31842.822} C_VEL
LIN {X 0,Y 680.471,Z 407.457,A -85,B 0,C 180,E1 31840.068,E2 31840.068} C_VEL
LIN {X 0,Y 680.525,Z 407.456,A -85,B 0,C 180,E1 31837.085,E2 31837.085} C_VEL
LIN {X 0,Y 680.458,Z 407.464,A -85,B 0,C 180,E1 31834.217,E2 31834.217} C_VEL
LIN {X 0,Y 680.531,Z 407.453,A -85,B 0,C 180,E1 31831.302,E2 31831.302} C_VEL
LIN {X 0,Y 680.504,Z 407.461,A -85,B 0,C 180,E1 31829.46,E2 31829.46} C_VEL
LIN {X 0,Y 679.573,Z 407.584,A -85,B 0,C 180,E1 31828.812,E2 31828.812} C_VEL
LIN {X 0,Y 673.077,Z 408.391,A -85,B 0,C 180,E1 31826.995,E2 31826.995} C_VEL
LIN {X 0,Y 672.526,Z 408.454,A -85,B 0,C 180,E1 31826.522,E2 31826.522} C_VEL
LIN {X 0,Y 672.507,Z 408.452,A -85,B 0,C 180,E1 31823.929,E2 31823.929} C_VEL
LIN {X 0,Y 672.594,Z 408.454,A -85,B 0,C 180,E1 31821.033,E2 31821.033} C_VEL
LIN {X 0,Y 672.493,Z 408.419,A -85,B 0,C 180,E1 31818.118,E2 31818.118} C_VEL
LIN {X 0,Y 672.51,Z 408.453,A -85,B 0,C 180,E1 31815.534,E2 31815.534} C_VEL
LIN {X 0,Y 672.502,Z 408.421,A -85,B 0,C 180,E1 31812.34,E2 31812.34} C_VEL
LIN {X 0,Y 672.482,Z 408.461,A -85,B 0,C 180,E1 31809.761,E2 31809.761} C_VEL
LIN {X 0,Y 672.544,Z 408.439,A -85,B 0,C 180,E1 31807.023,E2 31807.023} C_VEL
LIN {X 0,Y 672.554,Z 408.734,A -85,B 0,C 180,E1 31805.229,E2 31805.229} C_VEL
LIN {X 0,Y 674.911,Z 414.929,A -85,B 0,C 180,E1 31804.54,E2 31804.54} C_VEL
LIN {X 0,Y 686.26,Z 434.623,A -85,B 0,C 180,E1 31803.549,E2 31803.549} C_VEL
LIN {X 0,Y 687.179,Z 436.806,A -85,B 0,C 180,E1 31803.463,E2 31803.463} C_VEL
LIN {X 0,Y 684.801,Z 685.453,A -85,B 0,C 180,E1 31800.484,E2 31800.484} C_VEL
LIN {X 0,Y 683.693,Z 803.529,A -85,B 0,C 180,E1 31799.072,E2 31799.072} C_VEL
LIN {X 0,Y 683.098,Z 828.93,A -85,B 0,C 180,E1 31798.618,E2 31798.618} C_VEL
LIN {X 0,Y 682.419,Z 850.466,A -85,B 0,C 180,E1 31798.098,E2 31798.098} C_VEL
LIN {X 0,Y 681.565,Z 875.245,A -85,B 0,C 180,E1 31797.335,E2 31797.335} C_VEL
LIN {X 0,Y 680.703,Z 895.655,A -85,B 0,C 180,E1 31796.565,E2 31796.565} C_VEL
LIN {X 0,Y 679.719,Z 917.936,A -85,B 0,C 180,E1 31795.579,E2 31795.579} C_VEL
LIN {X 0,Y 678.616,Z 940.018,A -85,B 0,C 180,E1 31794.414,E2 31794.414} C_VEL
LIN {X 0,Y 677.605,Z 960.522,A -85,B 0,C 180,E1 31793.173,E2 31793.173} C_VEL
LIN {X 0,Y 676.541,Z 980.41,A -85,B 0,C 180,E1 31791.775,E2 31791.775} C_VEL
LIN {X 0,Y 675.614,Z 999.407,A -85,B 0,C 180,E1 31790.262,E2 31790.262} C_VEL
LIN {X 0,Y 674.74,Z 1016.775,A -85,B 0,C 180,E1 31788.668,E2 31788.668} C_VEL
LIN {X 0,Y 674.028,Z 1032.991,A -85,B 0,C 180,E1 31786.992,E2 31786.992} C_VEL
LIN {X 0,Y 673.406,Z 1047.736,A -85,B 0,C 180,E1 31785.237,E2 31785.237} C_VEL
LIN {X 0,Y 672.907,Z 1061.326,A -85,B 0,C 180,E1 31783.403,E2 31783.403} C_VEL
LIN {X 0,Y 672.52,Z 1073.412,A -85,B 0,C 180,E1 31781.492,E2 31781.492} C_VEL
LIN {X 0,Y 672.253,Z 1084.273,A -85,B 0,C 180,E1 31779.503,E2 31779.503} C_VEL
LIN {X 0,Y 672.093,Z 1093.152,A -85,B 0,C 180,E1 31777.523,E2 31777.523} C_VEL
LIN {X 0,Y 671.971,Z 1100.502,A -85,B 0,C 180,E1 31775.55,E2 31775.55} C_VEL
LIN {X 0,Y 671.911,Z 1106.365,A -85,B 0,C 180,E1 31773.498,E2 31773.498} C_VEL
LIN {X 0,Y 671.921,Z 1110.187,A -85,B 0,C 180,E1 31771.706,E2 31771.706} C_VEL
LIN {X 0,Y 671.909,Z 1113.178,A -85,B 0,C 180,E1 31769.574,E2 31769.574} C_VEL
LIN {X 0,Y 671.898,Z 1114.313,A -85,B 0,C 180,E1 31767.697,E2 31767.697} C_VEL
LIN {X 0,Y 671.91,Z 1114.208,A -85,B 0,C 180,E1 31765.818,E2 31765.818} C_VEL
LIN {X 0,Y 671.918,Z 1112.414,A -85,B 0,C 180,E1 31763.678,E2 31763.678} C_VEL
LIN {X 0,Y 671.925,Z 1109.572,A -85,B 0,C 180,E1 31761.873,E2 31761.873} C_VEL
LIN {X 0,Y 671.956,Z 1104.838,A -85,B 0,C 180,E1 31759.8,E2 31759.8} C_VEL
LIN {X 0,Y 671.997,Z 1098.69,A -85,B 0,C 180,E1 31757.845,E2 31757.845} C_VEL
LIN {X 0,Y 672.111,Z 1091.428,A -85,B 0,C 180,E1 31755.966,E2 31755.966} C_VEL
LIN {X 0,Y 672.322,Z 1081.588,A -85,B 0,C 180,E1 31753.894,E2 31753.894} C_VEL
LIN {X 0,Y 672.569,Z 1071.923,A -85,B 0,C 180,E1 31752.166,E2 31752.166} C_VEL
LIN {X 0,Y 673.001,Z 1058.49,A -85,B 0,C 180,E1 31750.109,E2 31750.109} C_VEL
LIN {X 0,Y 673.475,Z 1045.54,A -85,B 0,C 180,E1 31748.395,E2 31748.395} C_VEL
LIN {X 0,Y 674.202,Z 1028.977,A -85,B 0,C 180,E1 31746.488,E2 31746.488} C_VEL
LIN {X 0,Y 674.886,Z 1013.803,A -85,B 0,C 180,E1 31744.954,E2 31744.954} C_VEL
LIN {X 0,Y 675.826,Z 994.846,A -85,B 0,C 180,E1 31743.271,E2 31743.271} C_VEL
LIN {X 0,Y 676.722,Z 976.979,A -85,B 0,C 180,E1 31741.879,E2 31741.879} C_VEL
LIN {X 0,Y 677.83,Z 955.701,A -85,B 0,C 180,E1 31740.433,E2 31740.433} C_VEL
LIN {X 0,Y 678.813,Z 935.851,A -85,B 0,C 180,E1 31739.261,E2 31739.261} C_VEL
LIN {X 0,Y 679.96,Z 912.623,A -85,B 0,C 180,E1 31738.086,E2 31738.086} C_VEL
LIN {X 0,Y 680.815,Z 892.934,A -85,B 0,C 180,E1 31737.234,E2 31737.234} C_VEL
LIN {X 0,Y 681.798,Z 868.893,A -85,B 0,C 180,E1 31736.361,E2 31736.361} C_VEL
LIN {X 0,Y 682.551,Z 847.069,A -85,B 0,C 180,E1 31735.723,E2 31735.723} C_VEL
LIN {X 0,Y 683.292,Z 823.009,A -85,B 0,C 180,E1 31735.167,E2 31735.167} C_VEL
LIN {X 0,Y 683.732,Z 799.289,A -85,B 0,C 180,E1 31734.779,E2 31734.779} C_VEL
LIN {X 0,Y 686.027,Z 552.455,A -85,B 0,C 180,E1 31731.842,E2 31731.842} C_VEL
LIN {X 0,Y 687.029,Z 436.005,A -85,B 0,C 180,E1 31730.427,E2 31730.427} C_VEL
LIN {X 0,Y 677.128,Z 418.78,A -85,B 0,C 180,E1 31729.572,E2 31729.572} C_VEL
LIN {X 0,Y 674.507,Z 414.166,A -85,B 0,C 180,E1 31729.304,E2 31729.304} C_VEL
LIN {X 0,Y 672.535,Z 408.623,A -85,B 0,C 180,E1 31728.647,E2 31728.647} C_VEL
LIN {X 0,Y 672.485,Z 408.464,A -85,B 0,C 180,E1 31726.023,E2 31726.023} C_VEL
LIN {X 0,Y 672.55,Z 408.447,A -85,B 0,C 180,E1 31723.24,E2 31723.24} C_VEL
LIN {X 0,Y 672.505,Z 408.452,A -85,B 0,C 180,E1 31720.294,E2 31720.294} C_VEL
LIN {X 0,Y 672.499,Z 408.454,A -85,B 0,C 180,E1 31717.86,E2 31717.86} C_VEL
LIN {X 0,Y 672.573,Z 408.426,A -85,B 0,C 180,E1 31715,E2 31715} C_VEL
LIN {X 0,Y 672.511,Z 408.452,A -85,B 0,C 180,E1 31712.059,E2 31712.059} C_VEL
LIN {X 0,Y 672.518,Z 408.42,A -85,B 0,C 180,E1 31709.481,E2 31709.481} C_VEL
LIN {X 0,Y 672.558,Z 408.451,A -85,B 0,C 180,E1 31706.393,E2 31706.393} C_VEL
LIN {X 0,Y 672.519,Z 408.446,A -85,B 0,C 180,E1 31703.668,E2 31703.668} C_VEL
LIN {X 0,Y 672.588,Z 408.444,A -85,B 0,C 180,E1 31700.812,E2 31700.812} C_VEL
LIN {X 0,Y 672.533,Z 408.451,A -85,B 0,C 180,E1 31697.835,E2 31697.835} C_VEL
LIN {X 0,Y 672.566,Z 408.445,A -85,B 0,C 180,E1 31694.992,E2 31694.992} C_VEL
LIN {X 0,Y 672.549,Z 408.442,A -85,B 0,C 180,E1 31691.926,E2 31691.926} C_VEL
LIN {X 0,Y 672.558,Z 408.454,A -85,B 0,C 180,E1 31689.067,E2 31689.067} C_VEL
LIN {X 0,Y 672.562,Z 408.443,A -85,B 0,C 180,E1 31685.888,E2 31685.888} C_VEL
LIN {X 0,Y 672.572,Z 408.448,A -85,B 0,C 180,E1 31682.897,E2 31682.897} C_VEL
LIN {X 0,Y 672.564,Z 408.446,A -85,B 0,C 180,E1 31679.744,E2 31679.744} C_VEL
LIN {X 0,Y 672.583,Z 408.442,A -85,B 0,C 180,E1 31676.676,E2 31676.676} C_VEL
LIN {X 0,Y 672.566,Z 408.443,A -85,B 0,C 180,E1 31673.598,E2 31673.598} C_VEL
LIN {X 0,Y 672.582,Z 408.454,A -85,B 0,C 180,E1 31670.588,E2 31670.588} C_VEL
LIN {X 0,Y 672.57,Z 408.436,A -85,B 0,C 180,E1 31667.464,E2 31667.464} C_VEL
LIN {X 0,Y 672.579,Z 408.447,A -85,B 0,C 180,E1 31664.441,E2 31664.441} C_VEL
LIN {X 0,Y 672.576,Z 408.446,A -85,B 0,C 180,E1 31661.359,E2 31661.359} C_VEL
LIN {X 0,Y 672.569,Z 408.439,A -85,B 0,C 180,E1 31658.307,E2 31658.307} C_VEL
LIN {X 0,Y 672.581,Z 408.447,A -85,B 0,C 180,E1 31655.278,E2 31655.278} C_VEL
LIN {X 0,Y 672.565,Z 408.45,A -85,B 0,C 180,E1 31652.2,E2 31652.2} C_VEL
LIN {X 0,Y 672.585,Z 408.441,A -85,B 0,C 180,E1 31649.236,E2 31649.236} C_VEL
LIN {X 0,Y 672.56,Z 408.451,A -85,B 0,C 180,E1 31646.116,E2 31646.116} C_VEL
LIN {X 0,Y 672.585,Z 408.446,A -85,B 0,C 180,E1 31643.087,E2 31643.087} C_VEL
LIN {X 0,Y 672.554,Z 408.451,A -85,B 0,C 180,E1 31640.039,E2 31640.039} C_VEL
LIN {X 0,Y 672.578,Z 408.44,A -85,B 0,C 180,E1 31637.087,E2 31637.087} C_VEL
LIN {X 0,Y 672.547,Z 408.45,A -85,B 0,C 180,E1 31633.972,E2 31633.972} C_VEL
LIN {X 0,Y 672.585,Z 408.652,A -85,B 0,C 180,E1 31631.171,E2 31631.171} C_VEL
LIN {X 0,Y 678.894,Z 425.083,A -85,B 0,C 180,E1 31629.404,E2 31629.404} C_VEL
LIN {X 0,Y 682.835,Z 435.888,A -85,B 0,C 180,E1 31628.321,E2 31628.321} C_VEL
LIN {X 0,Y 682.385,Z 452.787,A -85,B 0,C 180,E1 31627.109,E2 31627.109} C_VEL
LIN {X 0,Y 687.146,Z 473.534,A -85,B 0,C 180,E1 31626.543,E2 31626.543} C_VEL
LIN {X 0,Y 684.844,Z 719.615,A -85,B 0,C 180,E1 31623.599,E2 31623.599} C_VEL
LIN {X 0,Y 683.704,Z 843.354,A -85,B 0,C 180,E1 31622.119,E2 31622.119} C_VEL
LIN {X 0,Y 683.096,Z 868.876,A -85,B 0,C 180,E1 31621.664,E2 31621.664} C_VEL
LIN {X 0,Y 682.419,Z 890.331,A -85,B 0,C 180,E1 31621.146,E2 31621.146} C_VEL
LIN {X 0,Y 681.597,Z 914.545,A -85,B 0,C 180,E1 31620.405,E2 31620.405} C_VEL
LIN {X 0,Y 680.719,Z 935.343,A -85,B 0,C 180,E1 31619.622,E2 31619.622} C_VEL
LIN {X 0,Y 679.794,Z 956.262,A -85,B 0,C 180,E1 31618.701,E2 31618.701} C_VEL
LIN {X 0,Y 678.692,Z 978.314,A -85,B 0,C 180,E1 31617.555,E2 31617.555} C_VEL
LIN {X 0,Y 677.758,Z 997.214,A -85,B 0,C 180,E1 31616.426,E2 31616.426} C_VEL
LIN {X 0,Y 676.662,Z 1018.006,A -85,B 0,C 180,E1 31615,E2 31615} C_VEL
LIN {X 0,Y 675.802,Z 1035.398,A -85,B 0,C 180,E1 31613.638,E2 31613.638} C_VEL
LIN {X 0,Y 674.848,Z 1054.604,A -85,B 0,C 180,E1 31611.924,E2 31611.924} C_VEL
LIN {X 0,Y 674.159,Z 1069.747,A -85,B 0,C 180,E1 31610.386,E2 31610.386} C_VEL
LIN {X 0,Y 673.468,Z 1085.815,A -85,B 0,C 180,E1 31608.525,E2 31608.525} C_VEL
LIN {X 0,Y 673.008,Z 1098.525,A -85,B 0,C 180,E1 31606.841,E2 31606.841} C_VEL
LIN {X 0,Y 672.589,Z 1111.763,A -85,B 0,C 180,E1 31604.815,E2 31604.815} C_VEL
LIN {X 0,Y 672.316,Z 1121.605,A -85,B 0,C 180,E1 31603.058,E2 31603.058} C_VEL
LIN {X 0,Y 672.102,Z 1131.476,A -85,B 0,C 180,E1 31600.978,E2 31600.978} C_VEL
LIN {X 0,Y 672.004,Z 1138.514,A -85,B 0,C 180,E1 31599.161,E2 31599.161} C_VEL
LIN {X 0,Y 671.934,Z 1144.507,A -85,B 0,C 180,E1 31597.267,E2 31597.267} C_VEL
LIN {X 0,Y 671.893,Z 1149.337,A -85,B 0,C 180,E1 31595.208,E2 31595.208} C_VEL
LIN {X 0,Y 671.908,Z 1152.237,A -85,B 0,C 180,E1 31593.413,E2 31593.413} C_VEL
LIN {X 0,Y 671.907,Z 1154.17,A -85,B 0,C 180,E1 31591.279,E2 31591.279} C_VEL
LIN {X 0,Y 671.882,Z 1154.351,A -85,B 0,C 180,E1 31589.403,E2 31589.403} C_VEL
LIN {X 0,Y 671.907,Z 1153.363,A -85,B 0,C 180,E1 31587.612,E2 31587.612} C_VEL
LIN {X 0,Y 671.918,Z 1150.449,A -85,B 0,C 180,E1 31585.391,E2 31585.391} C_VEL
LIN {X 0,Y 671.93,Z 1146.689,A -85,B 0,C 180,E1 31583.592,E2 31583.592} C_VEL
LIN {X 0,Y 671.983,Z 1141.201,A -85,B 0,C 180,E1 31581.615,E2 31581.615} C_VEL
LIN {X 0,Y 672.088,Z 1133.604,A -85,B 0,C 180,E1 31579.543,E2 31579.543} C_VEL
LIN {X 0,Y 672.243,Z 1125.118,A -85,B 0,C 180,E1 31577.632,E2 31577.632} C_VEL
LIN {X 0,Y 672.508,Z 1114.353,A -85,B 0,C 180,E1 31575.623,E2 31575.623} C_VEL
LIN {X 0,Y 672.841,Z 1103.388,A -85,B 0,C 180,E1 31573.865,E2 31573.865} C_VEL
LIN {X 0,Y 673.362,Z 1088.942,A -85,B 0,C 180,E1 31571.87,E2 31571.87} C_VEL
LIN {X 0,Y 673.937,Z 1074.714,A -85,B 0,C 180,E1 31570.16,E2 31570.16} C_VEL
LIN {X 0,Y 674.683,Z 1058.309,A -85,B 0,C 180,E1 31568.436,E2 31568.436} C_VEL
LIN {X 0,Y 675.451,Z 1042.138,A -85,B 0,C 180,E1 31566.935,E2 31566.935} C_VEL
LIN {X 0,Y 676.436,Z 1022.867,A -85,B 0,C 180,E1 31565.364,E2 31565.364} C_VEL
LIN {X 0,Y 677.326,Z 1005.07,A -85,B 0,C 180,E1 31564.089,E2 31564.089} C_VEL
LIN {X 0,Y 678.488,Z 982.882,A -85,B 0,C 180,E1 31562.704,E2 31562.704} C_VEL
LIN {X 0,Y 679.432,Z 963.336,A -85,B 0,C 180,E1 31561.649,E2 31561.649} C_VEL
LIN {X 0,Y 680.535,Z 939.862,A -85,B 0,C 180,E1 31560.563,E2 31560.563} C_VEL
LIN {X 0,Y 681.373,Z 919.683,A -85,B 0,C 180,E1 31559.779,E2 31559.779} C_VEL
LIN {X 0,Y 682.248,Z 897.147,A -85,B 0,C 180,E1 31559.041,E2 31559.041} C_VEL
LIN {X 0,Y 682.94,Z 873.134,A -85,B 0,C 180,E1 31558.428,E2 31558.428} C_VEL
LIN {X 0,Y 683.576,Z 850.383,A -85,B 0,C 180,E1 31557.987,E2 31557.987} C_VEL
LIN {X 0,Y 684,Z 816.682,A -85,B 0,C 180,E1 31557.545,E2 31557.545} C_VEL
LIN {X 0,Y 686.029,Z 585.709,A -85,B 0,C 180,E1 31554.804,E2 31554.804} C_VEL
LIN {X 0,Y 686.966,Z 471.98,A -85,B 0,C 180,E1 31553.426,E2 31553.426} C_VEL
LIN {X 0,Y 682.333,Z 452.185,A -85,B 0,C 180,E1 31552.861,E2 31552.861} C_VEL
LIN {X 0,Y 682.662,Z 435.135,A -85,B 0,C 180,E1 31551.608,E2 31551.608} C_VEL
LIN {X 0,Y 673.736,Z 411.737,A -85,B 0,C 180,E1 31549.191,E2 31549.191} C_VEL
LIN {X 0,Y 672.576,Z 408.596,A -85,B 0,C 180,E1 31548.807,E2 31548.807} C_VEL
LIN {X 0,Y 672.556,Z 408.448,A -85,B 0,C 180,E1 31545.896,E2 31545.896} C_VEL
LIN {X 0,Y 672.562,Z 408.429,A -85,B 0,C 180,E1 31542.741,E2 31542.741} C_VEL
LIN {X 0,Y 672.568,Z 408.437,A -85,B 0,C 180,E1 31539.738,E2 31539.738} C_VEL
LIN {X 0,Y 672.567,Z 408.439,A -85,B 0,C 180,E1 31536.595,E2 31536.595} C_VEL
LIN {X 0,Y 672.582,Z 408.446,A -85,B 0,C 180,E1 31533.575,E2 31533.575} C_VEL
LIN {X 0,Y 672.568,Z 408.448,A -85,B 0,C 180,E1 31530.427,E2 31530.427} C_VEL
LIN {X 0,Y 672.584,Z 408.448,A -85,B 0,C 180,E1 31527.436,E2 31527.436} C_VEL
LIN {X 0,Y 672.571,Z 408.437,A -85,B 0,C 180,E1 31524.31,E2 31524.31} C_VEL
LIN {X 0,Y 672.58,Z 408.452,A -85,B 0,C 180,E1 31521.269,E2 31521.269} C_VEL
LIN {X 0,Y 672.574,Z 408.44,A -85,B 0,C 180,E1 31518.192,E2 31518.192} C_VEL
LIN {X 0,Y 672.573,Z 408.444,A -85,B 0,C 180,E1 31515.168,E2 31515.168} C_VEL
LIN {X 0,Y 672.579,Z 408.444,A -85,B 0,C 180,E1 31512.1,E2 31512.1} C_VEL
LIN {X 0,Y 672.568,Z 408.44,A -85,B 0,C 180,E1 31509.067,E2 31509.067} C_VEL
LIN {X 0,Y 672.586,Z 408.445,A -85,B 0,C 180,E1 31506.059,E2 31506.059} C_VEL
LIN {X 0,Y 672.562,Z 408.443,A -85,B 0,C 180,E1 31502.983,E2 31502.983} C_VEL
LIN {X 0,Y 672.588,Z 408.445,A -85,B 0,C 180,E1 31499.915,E2 31499.915} C_VEL
LIN {X 0,Y 672.554,Z 408.448,A -85,B 0,C 180,E1 31496.847,E2 31496.847} C_VEL
LIN {X 0,Y 672.586,Z 408.445,A -85,B 0,C 180,E1 31493.855,E2 31493.855} C_VEL
LIN {X 0,Y 672.548,Z 408.451,A -85,B 0,C 180,E1 31490.76,E2 31490.76} C_VEL
LIN {X 0,Y 672.576,Z 408.445,A -85,B 0,C 180,E1 31487.813,E2 31487.813} C_VEL
LIN {X 0,Y 672.546,Z 408.454,A -85,B 0,C 180,E1 31484.743,E2 31484.743} C_VEL
LIN {X 0,Y 672.551,Z 408.444,A -85,B 0,C 180,E1 31481.897,E2 31481.897} C_VEL
LIN {X 0,Y 672.543,Z 408.454,A -85,B 0,C 180,E1 31478.73,E2 31478.73} C_VEL
LIN {X 0,Y 672.525,Z 408.438,A -85,B 0,C 180,E1 31476.053,E2 31476.053} C_VEL
LIN {X 0,Y 672.58,Z 408.452,A -85,B 0,C 180,E1 31473.036,E2 31473.036} C_VEL
LIN {X 0,Y 672.513,Z 408.453,A -85,B 0,C 180,E1 31470.225,E2 31470.225} C_VEL
LIN {X 0,Y 672.546,Z 408.449,A -85,B 0,C 180,E1 31467.54,E2 31467.54} C_VEL
LIN {X 0,Y 672.526,Z 408.454,A -85,B 0,C 180,E1 31466.522,E2 31466.522} C_VEL
LIN {X 0,Y 671.518,Z 408.58,A -85,B 0,C 180,E1 31465.866,E2 31465.866} C_VEL
LIN {X 0,Y 665.087,Z 409.378,A -85,B 0,C 180,E1 31464.027,E2 31464.027} C_VEL
LIN {X 0,Y 664.593,Z 409.439,A -85,B 0,C 180,E1 31463.548,E2 31463.548} C_VEL
LIN {X 0,Y 664.581,Z 409.44,A -85,B 0,C 180,E1 31460.474,E2 31460.474} C_VEL
LIN {X 0,Y 664.555,Z 409.404,A -85,B 0,C 180,E1 31457.851,E2 31457.851} C_VEL
LIN {X 0,Y 664.636,Z 409.445,A -85,B 0,C 180,E1 31454.876,E2 31454.876} C_VEL
LIN {X 0,Y 664.544,Z 409.407,A -85,B 0,C 180,E1 31451.988,E2 31451.988} C_VEL
LIN {X 0,Y 664.562,Z 409.451,A -85,B 0,C 180,E1 31449.415,E2 31449.415} C_VEL
LIN {X 0,Y 664.561,Z 409.451,A -85,B 0,C 180,E1 31446.248,E2 31446.248} C_VEL
LIN {X 0,Y 664.596,Z 409.807,A -85,B 0,C 180,E1 31445.7,E2 31445.7} C_VEL
LIN {X 0,Y 666.707,Z 415.288,A -85,B 0,C 180,E1 31445.085,E2 31445.085} C_VEL
LIN {X 0,Y 680.037,Z 437.919,A -85,B 0,C 180,E1 31443.9,E2 31443.9} C_VEL
LIN {X 0,Y 680.734,Z 439.815,A -85,B 0,C 180,E1 31443.831,E2 31443.831} C_VEL
LIN {X 0,Y 678.103,Z 688.33,A -85,B 0,C 180,E1 31440.824,E2 31440.824} C_VEL
LIN {X 0,Y 676.908,Z 803.663,A -85,B 0,C 180,E1 31439.432,E2 31439.432} C_VEL
LIN {X 0,Y 676.264,Z 829.013,A -85,B 0,C 180,E1 31438.974,E2 31438.974} C_VEL
LIN {X 0,Y 675.541,Z 850.216,A -85,B 0,C 180,E1 31438.458,E2 31438.458} C_VEL
LIN {X 0,Y 674.648,Z 873.806,A -85,B 0,C 180,E1 31437.735,E2 31437.735} C_VEL
LIN {X 0,Y 673.699,Z 894.281,A -85,B 0,C 180,E1 31436.963,E2 31436.963} C_VEL
LIN {X 0,Y 672.718,Z 914.907,A -85,B 0,C 180,E1 31436.054,E2 31436.054} C_VEL
LIN {X 0,Y 671.47,Z 937.553,A -85,B 0,C 180,E1 31434.877,E2 31434.877} C_VEL
LIN {X 0,Y 670.398,Z 957.392,A -85,B 0,C 180,E1 31433.683,E2 31433.683} C_VEL
LIN {X 0,Y 669.171,Z 978.541,A -85,B 0,C 180,E1 31432.212,E2 31432.212} C_VEL
LIN {X 0,Y 668.217,Z 995.878,A -85,B 0,C 180,E1 31430.838,E2 31430.838} C_VEL
LIN {X 0,Y 667.199,Z 1014.44,A -85,B 0,C 180,E1 31429.16,E2 31429.16} C_VEL
LIN {X 0,Y 666.453,Z 1029.245,A -85,B 0,C 180,E1 31427.642,E2 31427.642} C_VEL
LIN {X 0,Y 665.645,Z 1045.959,A -85,B 0,C 180,E1 31425.687,E2 31425.687} C_VEL
LIN {X 0,Y 665.141,Z 1058.487,A -85,B 0,C 180,E1 31424.006,E2 31424.006} C_VEL
LIN {X 0,Y 664.67,Z 1071.584,A -85,B 0,C 180,E1 31421.982,E2 31421.982} C_VEL
LIN {X 0,Y 664.373,Z 1081.606,A -85,B 0,C 180,E1 31420.171,E2 31420.171} C_VEL
LIN {X 0,Y 664.139,Z 1091.544,A -85,B 0,C 180,E1 31418.049,E2 31418.049} C_VEL
LIN {X 0,Y 664.027,Z 1098.52,A -85,B 0,C 180,E1 31416.224,E2 31416.224} C_VEL
LIN {X 0,Y 663.955,Z 1104.734,A -85,B 0,C 180,E1 31414.232,E2 31414.232} C_VEL
LIN {X 0,Y 663.923,Z 1109.462,A -85,B 0,C 180,E1 31412.158,E2 31412.158} C_VEL
LIN {X 0,Y 663.923,Z 1112.43,A -85,B 0,C 180,E1 31410.259,E2 31410.259} C_VEL
LIN {X 0,Y 663.912,Z 1114.231,A -85,B 0,C 180,E1 31408.015,E2 31408.015} C_VEL
LIN {X 0,Y 663.895,Z 1114.312,A -85,B 0,C 180,E1 31406.2,E2 31406.2} C_VEL
LIN {X 0,Y 663.908,Z 1113.033,A -85,B 0,C 180,E1 31404.122,E2 31404.122} C_VEL
LIN {X 0,Y 663.922,Z 1109.984,A -85,B 0,C 180,E1 31402.036,E2 31402.036} C_VEL
LIN {X 0,Y 663.929,Z 1106.052,A -85,B 0,C 180,E1 31400.202,E2 31400.202} C_VEL
LIN {X 0,Y 663.988,Z 1099.635,A -85,B 0,C 180,E1 31398.006,E2 31398.006} C_VEL
LIN {X 0,Y 664.116,Z 1092.711,A -85,B 0,C 180,E1 31396.149,E2 31396.149} C_VEL
LIN {X 0,Y 664.333,Z 1083.494,A -85,B 0,C 180,E1 31394.102,E2 31394.102} C_VEL
LIN {X 0,Y 664.605,Z 1073.274,A -85,B 0,C 180,E1 31392.217,E2 31392.217} C_VEL
LIN {X 0,Y 665.045,Z 1060.967,A -85,B 0,C 180,E1 31390.253,E2 31390.253} C_VEL
LIN {X 0,Y 665.588,Z 1047.378,A -85,B 0,C 180,E1 31388.404,E2 31388.404} C_VEL
LIN {X 0,Y 666.295,Z 1032.871,A -85,B 0,C 180,E1 31386.66,E2 31386.66} C_VEL
LIN {X 0,Y 667.072,Z 1016.686,A -85,B 0,C 180,E1 31384.971,E2 31384.971} C_VEL
LIN {X 0,Y 668.043,Z 999.395,A -85,B 0,C 180,E1 31383.367,E2 31383.367} C_VEL
LIN {X 0,Y 669.044,Z 980.646,A -85,B 0,C 180,E1 31381.856,E2 31381.856} C_VEL
LIN {X 0,Y 670.236,Z 960.579,A -85,B 0,C 180,E1 31380.43,E2 31380.43} C_VEL
LIN {X 0,Y 671.336,Z 940.123,A -85,B 0,C 180,E1 31379.179,E2 31379.179} C_VEL
LIN {X 0,Y 672.514,Z 918.801,A -85,B 0,C 180,E1 31378.042,E2 31378.042} C_VEL
LIN {X 0,Y 673.6,Z 896.578,A -85,B 0,C 180,E1 31377.041,E2 31377.041} C_VEL
LIN {X 0,Y 674.495,Z 877.128,A -85,B 0,C 180,E1 31376.295,E2 31376.295} C_VEL
LIN {X 0,Y 675.474,Z 852.055,A -85,B 0,C 180,E1 31375.501,E2 31375.501} C_VEL
LIN {X 0,Y 676.209,Z 830.424,A -85,B 0,C 180,E1 31374.967,E2 31374.967} C_VEL
LIN {X 0,Y 676.889,Z 805.608,A -85,B 0,C 180,E1 31374.506,E2 31374.506} C_VEL
LIN {X 0,Y 677.529,Z 747.152,A -85,B 0,C 180,E1 31373.786,E2 31373.786} C_VEL
LIN {X 0,Y 680.052,Z 501.871,A -85,B 0,C 180,E1 31370.837,E2 31370.837} C_VEL
LIN {X 0,Y 680.602,Z 439.033,A -85,B 0,C 180,E1 31370.061,E2 31370.061} C_VEL
LIN {X 0,Y 669.004,Z 419.125,A -85,B 0,C 180,E1 31369.038,E2 31369.038} C_VEL
LIN {X 0,Y 666.67,Z 415.212,A -85,B 0,C 180,E1 31368.82,E2 31368.82} C_VEL
LIN {X 0,Y 664.567,Z 409.628,A -85,B 0,C 180,E1 31368.167,E2 31368.167} C_VEL
LIN {X 0,Y 664.558,Z 409.452,A -85,B 0,C 180,E1 31365.722,E2 31365.722} C_VEL
LIN {X 0,Y 664.588,Z 409.421,A -85,B 0,C 180,E1 31362.613,E2 31362.613} C_VEL
LIN {X 0,Y 664.556,Z 409.442,A -85,B 0,C 180,E1 31359.976,E2 31359.976} C_VEL
LIN {X 0,Y 664.586,Z 409.424,A -85,B 0,C 180,E1 31357.402,E2 31357.402} C_VEL
LIN {X 0,Y 664.579,Z 409.441,A -85,B 0,C 180,E1 31354.243,E2 31354.243} C_VEL
LIN {X 0,Y 664.576,Z 409.441,A -85,B 0,C 180,E1 31351.573,E2 31351.573} C_VEL
LIN {X 0,Y 664.628,Z 409.416,A -85,B 0,C 180,E1 31348.527,E2 31348.527} C_VEL
LIN {X 0,Y 664.579,Z 409.444,A -85,B 0,C 180,E1 31345.678,E2 31345.678} C_VEL
LIN {X 0,Y 664.653,Z 409.442,A -85,B 0,C 180,E1 31342.745,E2 31342.745} C_VEL
LIN {X 0,Y 664.587,Z 409.432,A -85,B 0,C 180,E1 31339.787,E2 31339.787} C_VEL
LIN {X 0,Y 664.64,Z 409.436,A -85,B 0,C 180,E1 31336.879,E2 31336.879} C_VEL
LIN {X 0,Y 664.602,Z 409.439,A -85,B 0,C 180,E1 31333.84,E2 31333.84} C_VEL
LIN {X 0,Y 664.631,Z 409.432,A -85,B 0,C 180,E1 31330.927,E2 31330.927} C_VEL
LIN {X 0,Y 664.611,Z 409.434,A -85,B 0,C 180,E1 31327.782,E2 31327.782} C_VEL
LIN {X 0,Y 664.639,Z 409.441,A -85,B 0,C 180,E1 31324.833,E2 31324.833} C_VEL
LIN {X 0,Y 664.619,Z 409.425,A -85,B 0,C 180,E1 31321.724,E2 31321.724} C_VEL
LIN {X 0,Y 664.645,Z 409.436,A -85,B 0,C 180,E1 31318.707,E2 31318.707} C_VEL
LIN {X 0,Y 664.625,Z 409.433,A -85,B 0,C 180,E1 31315.6,E2 31315.6} C_VEL
LIN {X 0,Y 664.645,Z 409.429,A -85,B 0,C 180,E1 31312.566,E2 31312.566} C_VEL
LIN {X 0,Y 664.626,Z 409.436,A -85,B 0,C 180,E1 31309.424,E2 31309.424} C_VEL
LIN {X 0,Y 664.637,Z 409.442,A -85,B 0,C 180,E1 31306.375,E2 31306.375} C_VEL
LIN {X 0,Y 664.629,Z 409.429,A -85,B 0,C 180,E1 31303.301,E2 31303.301} C_VEL
LIN {X 0,Y 664.632,Z 409.437,A -85,B 0,C 180,E1 31300.306,E2 31300.306} C_VEL
LIN {X 0,Y 664.636,Z 409.427,A -85,B 0,C 180,E1 31297.252,E2 31297.252} C_VEL
LIN {X 0,Y 664.628,Z 409.429,A -85,B 0,C 180,E1 31294.228,E2 31294.228} C_VEL
LIN {X 0,Y 664.645,Z 409.435,A -85,B 0,C 180,E1 31291.222,E2 31291.222} C_VEL
LIN {X 0,Y 664.621,Z 409.434,A -85,B 0,C 180,E1 31288.125,E2 31288.125} C_VEL
LIN {X 0,Y 664.644,Z 409.434,A -85,B 0,C 180,E1 31285.075,E2 31285.075} C_VEL
LIN {X 0,Y 664.614,Z 409.439,A -85,B 0,C 180,E1 31282.024,E2 31282.024} C_VEL
LIN {X 0,Y 664.647,Z 409.439,A -85,B 0,C 180,E1 31279.011,E2 31279.011} C_VEL
LIN {X 0,Y 664.609,Z 409.444,A -85,B 0,C 180,E1 31275.967,E2 31275.967} C_VEL
LIN {X 0,Y 664.642,Z 409.439,A -85,B 0,C 180,E1 31272.961,E2 31272.961} C_VEL
LIN {X 0,Y 664.632,Z 409.688,A -85,B 0,C 180,E1 31271.662,E2 31271.662} C_VEL
LIN {X 0,Y 671.499,Z 427.565,A -85,B 0,C 180,E1 31269.703,E2 31269.703} C_VEL
LIN {X 0,Y 675.806,Z 439.471,A -85,B 0,C 180,E1 31268.493,E2 31268.493} C_VEL
LIN {X 0,Y 675.427,Z 452.298,A -85,B 0,C 180,E1 31267.564,E2 31267.564} C_VEL
LIN {X 0,Y 680.674,Z 475.295,A -85,B 0,C 180,E1 31266.922,E2 31266.922} C_VEL
LIN {X 0,Y 678.167,Z 720.887,A -85,B 0,C 180,E1 31263.959,E2 31263.959} C_VEL
LIN {X 0,Y 676.919,Z 843.502,A -85,B 0,C 180,E1 31262.478,E2 31262.478} C_VEL
LIN {X 0,Y 676.261,Z 869.005,A -85,B 0,C 180,E1 31262.019,E2 31262.019} C_VEL
LIN {X 0,Y 675.536,Z 890.221,A -85,B 0,C 180,E1 31261.503,E2 31261.503} C_VEL
LIN {X 0,Y 674.678,Z 913.257,A -85,B 0,C 180,E1 31260.8,E2 31260.8} C_VEL
LIN {X 0,Y 673.707,Z 934.207,A -85,B 0,C 180,E1 31260.011,E2 31260.011} C_VEL
LIN {X 0,Y 672.747,Z 954.27,A -85,B 0,C 180,E1 31259.128,E2 31259.128} C_VEL
LIN {X 0,Y 671.476,Z 977.499,A -85,B 0,C 180,E1 31257.925,E2 31257.925} C_VEL
LIN {X 0,Y 670.428,Z 996.729,A -85,B 0,C 180,E1 31256.77,E2 31256.77} C_VEL
LIN {X 0,Y 669.207,Z 1018.004,A -85,B 0,C 180,E1 31255.298,E2 31255.298} C_VEL
LIN {X 0,Y 668.242,Z 1035.399,A -85,B 0,C 180,E1 31253.922,E2 31253.922} C_VEL
LIN {X 0,Y 667.193,Z 1054.604,A -85,B 0,C 180,E1 31252.189,E2 31252.189} C_VEL
LIN {X 0,Y 666.423,Z 1069.631,A -85,B 0,C 180,E1 31250.646,E2 31250.646} C_VEL
LIN {X 0,Y 665.653,Z 1085.817,A -85,B 0,C 180,E1 31248.751,E2 31248.751} C_VEL
LIN {X 0,Y 665.146,Z 1098.539,A -85,B 0,C 180,E1 31247.044,E2 31247.044} C_VEL
LIN {X 0,Y 664.67,Z 1111.764,A -85,B 0,C 180,E1 31244.996,E2 31244.996} C_VEL
LIN {X 0,Y 664.356,Z 1121.945,A -85,B 0,C 180,E1 31243.151,E2 31243.151} C_VEL
LIN {X 0,Y 664.118,Z 1131.956,A -85,B 0,C 180,E1 31240.993,E2 31240.993} C_VEL
LIN {X 0,Y 664.014,Z 1138.817,A -85,B 0,C 180,E1 31239.185,E2 31239.185} C_VEL
LIN {X 0,Y 663.949,Z 1145.244,A -85,B 0,C 180,E1 31237.094,E2 31237.094} C_VEL
LIN {X 0,Y 663.894,Z 1149.656,A -85,B 0,C 180,E1 31235.098,E2 31235.098} C_VEL
LIN {X 0,Y 663.898,Z 1152.462,A -85,B 0,C 180,E1 31233.281,E2 31233.281} C_VEL
LIN {X 0,Y 663.909,Z 1154.215,A -85,B 0,C 180,E1 31231.122,E2 31231.122} C_VEL
LIN {X 0,Y 663.884,Z 1154.328,A -85,B 0,C 180,E1 31229.31,E2 31229.31} C_VEL
LIN {X 0,Y 663.891,Z 1153.226,A -85,B 0,C 180,E1 31227.41,E2 31227.41} C_VEL
LIN {X 0,Y 663.91,Z 1150.291,A -85,B 0,C 180,E1 31225.249,E2 31225.249} C_VEL
LIN {X 0,Y 663.933,Z 1146.483,A -85,B 0,C 180,E1 31223.428,E2 31223.428} C_VEL
LIN {X 0,Y 663.984,Z 1140.635,A -85,B 0,C 180,E1 31221.339,E2 31221.339} C_VEL
LIN {X 0,Y 664.107,Z 1133.604,A -85,B 0,C 180,E1 31219.415,E2 31219.415} C_VEL
LIN {X 0,Y 664.289,Z 1125.119,A -85,B 0,C 180,E1 31217.482,E2 31217.482} C_VEL
LIN {X 0,Y 664.584,Z 1114.352,A -85,B 0,C 180,E1 31215.448,E2 31215.448} C_VEL
LIN {X 0,Y 664.952,Z 1103.389,A -85,B 0,C 180,E1 31213.669,E2 31213.669} C_VEL
LIN {X 0,Y 665.52,Z 1089.326,A -85,B 0,C 180,E1 31211.699,E2 31211.699} C_VEL
LIN {X 0,Y 666.109,Z 1076.081,A -85,B 0,C 180,E1 31210.077,E2 31210.077} C_VEL
LIN {X 0,Y 667.003,Z 1058.308,A -85,B 0,C 180,E1 31208.175,E2 31208.175} C_VEL
LIN {X 0,Y 667.854,Z 1042.291,A -85,B 0,C 180,E1 31206.671,E2 31206.671} C_VEL
LIN {X 0,Y 668.966,Z 1022.26,A -85,B 0,C 180,E1 31205.023,E2 31205.023} C_VEL
LIN {X 0,Y 670.026,Z 1003.731,A -85,B 0,C 180,E1 31203.69,E2 31203.69} C_VEL
LIN {X 0,Y 671.229,Z 982.362,A -85,B 0,C 180,E1 31202.353,E2 31202.353} C_VEL
LIN {X 0,Y 672.271,Z 962.749,A -85,B 0,C 180,E1 31201.288,E2 31201.288} C_VEL
LIN {X 0,Y 673.51,Z 938.732,A -85,B 0,C 180,E1 31200.176,E2 31200.176} C_VEL
LIN {X 0,Y 674.38,Z 919.679,A -85,B 0,C 180,E1 31199.432,E2 31199.432} C_VEL
LIN {X 0,Y 675.332,Z 896.983,A -85,B 0,C 180,E1 31198.683,E2 31198.683} C_VEL
LIN {X 0,Y 676.104,Z 873.051,A -85,B 0,C 180,E1 31198.069,E2 31198.069} C_VEL
LIN {X 0,Y 676.785,Z 850.382,A -85,B 0,C 180,E1 31197.627,E2 31197.627} C_VEL
LIN {X 0,Y 677.249,Z 816.625,A -85,B 0,C 180,E1 31197.181,E2 31197.181} C_VEL
LIN {X 0,Y 679.465,Z 586.193,A -85,B 0,C 180,E1 31194.422,E2 31194.422} C_VEL
LIN {X 0,Y 680.505,Z 473.775,A -85,B 0,C 180,E1 31193.048,E2 31193.048} C_VEL
LIN {X 0,Y 675.397,Z 451.883,A -85,B 0,C 180,E1 31192.414,E2 31192.414} C_VEL
LIN {X 0,Y 675.834,Z 439.057,A -85,B 0,C 180,E1 31191.474,E2 31191.474} C_VEL
LIN {X 0,Y 667.069,Z 415.974,A -85,B 0,C 180,E1 31189.066,E2 31189.066} C_VEL
LIN {X 0,Y 664.623,Z 409.637,A -85,B 0,C 180,E1 31188.347,E2 31188.347} C_VEL
LIN {X 0,Y 664.645,Z 409.432,A -85,B 0,C 180,E1 31185.487,E2 31185.487} C_VEL
LIN {X 0,Y 664.605,Z 409.409,A -85,B 0,C 180,E1 31182.494,E2 31182.494} C_VEL
LIN {X 0,Y 664.647,Z 409.428,A -85,B 0,C 180,E1 31179.488,E2 31179.488} C_VEL
LIN {X 0,Y 664.616,Z 409.429,A -85,B 0,C 180,E1 31176.4,E2 31176.4} C_VEL
LIN {X 0,Y 664.643,Z 409.431,A -85,B 0,C 180,E1 31173.39,E2 31173.39} C_VEL
LIN {X 0,Y 664.621,Z 409.439,A -85,B 0,C 180,E1 31170.281,E2 31170.281} C_VEL
LIN {X 0,Y 664.643,Z 409.44,A -85,B 0,C 180,E1 31167.313,E2 31167.313} C_VEL
LIN {X 0,Y 664.628,Z 409.426,A -85,B 0,C 180,E1 31164.25,E2 31164.25} C_VEL
LIN {X 0,Y 664.642,Z 409.44,A -85,B 0,C 180,E1 31161.258,E2 31161.258} C_VEL
LIN {X 0,Y 664.633,Z 409.429,A -85,B 0,C 180,E1 31158.145,E2 31158.145} C_VEL
LIN {X 0,Y 664.63,Z 409.431,A -85,B 0,C 180,E1 31155.086,E2 31155.086} C_VEL
LIN {X 0,Y 664.639,Z 409.433,A -85,B 0,C 180,E1 31152.07,E2 31152.07} C_VEL
LIN {X 0,Y 664.625,Z 409.427,A -85,B 0,C 180,E1 31149.002,E2 31149.002} C_VEL
LIN {X 0,Y 664.643,Z 409.435,A -85,B 0,C 180,E1 31145.958,E2 31145.958} C_VEL
LIN {X 0,Y 664.62,Z 409.431,A -85,B 0,C 180,E1 31142.932,E2 31142.932} C_VEL
LIN {X 0,Y 664.65,Z 409.435,A -85,B 0,C 180,E1 31139.914,E2 31139.914} C_VEL
LIN {X 0,Y 664.613,Z 409.436,A -85,B 0,C 180,E1 31136.809,E2 31136.809} C_VEL
LIN {X 0,Y 664.648,Z 409.435,A -85,B 0,C 180,E1 31133.782,E2 31133.782} C_VEL
LIN {X 0,Y 664.608,Z 409.44,A -85,B 0,C 180,E1 31130.732,E2 31130.732} C_VEL
LIN {X 0,Y 664.642,Z 409.434,A -85,B 0,C 180,E1 31127.753,E2 31127.753} C_VEL
LIN {X 0,Y 664.6,Z 409.442,A -85,B 0,C 180,E1 31124.645,E2 31124.645} C_VEL
LIN {X 0,Y 664.625,Z 409.432,A -85,B 0,C 180,E1 31121.764,E2 31121.764} C_VEL
LIN {X 0,Y 664.597,Z 409.443,A -85,B 0,C 180,E1 31118.637,E2 31118.637} C_VEL
LIN {X 0,Y 664.592,Z 409.426,A -85,B 0,C 180,E1 31115.938,E2 31115.938} C_VEL
LIN {X 0,Y 664.612,Z 409.438,A -85,B 0,C 180,E1 31112.783,E2 31112.783} C_VEL
LIN {X 0,Y 664.576,Z 409.441,A -85,B 0,C 180,E1 31110.069,E2 31110.069} C_VEL
LIN {X 0,Y 664.648,Z 409.431,A -85,B 0,C 180,E1 31107.106,E2 31107.106} C_VEL
LIN {X 0,Y 664.566,Z 409.441,A -85,B 0,C 180,E1 31104.177,E2 31104.177} C_VEL
LIN {X 0,Y 664.593,Z 409.439,A -85,B 0,C 180,E1 31103.548,E2 31103.548} C_VEL
LIN {X 0,Y 663.662,Z 409.562,A -85,B 0,C 180,E1 31102.884,E2 31102.884} C_VEL
LIN {X 0,Y 657.13,Z 410.378,A -85,B 0,C 180,E1 31100.975,E2 31100.975} C_VEL
LIN {X 0,Y 656.649,Z 410.429,A -85,B 0,C 180,E1 31100.539,E2 31100.539} C_VEL
LIN {X 0,Y 656.614,Z 410.39,A -85,B 0,C 180,E1 31097.868,E2 31097.868} C_VEL
LIN {X 0,Y 656.698,Z 410.433,A -85,B 0,C 180,E1 31094.926,E2 31094.926} C_VEL
LIN {X 0,Y 656.605,Z 410.393,A -85,B 0,C 180,E1 31091.953,E2 31091.953} C_VEL
LIN {X 0,Y 656.636,Z 410.44,A -85,B 0,C 180,E1 31089.306,E2 31089.306} C_VEL
LIN {X 0,Y 656.643,Z 410.595,A -85,B 0,C 180,E1 31086.242,E2 31086.242} C_VEL
LIN {X 0,Y 658.241,Z 415.186,A -85,B 0,C 180,E1 31085.684,E2 31085.684} C_VEL
LIN {X 0,Y 670.302,Z 435.115,A -85,B 0,C 180,E1 31084.571,E2 31084.571} C_VEL
LIN {X 0,Y 674.32,Z 442.565,A -85,B 0,C 180,E1 31084.208,E2 31084.208} C_VEL
LIN {X 0,Y 671.446,Z 691.19,A -85,B 0,C 180,E1 31081.173,E2 31081.173} C_VEL
LIN {X 0,Y 670.151,Z 804.782,A -85,B 0,C 180,E1 31079.786,E2 31079.786} C_VEL
LIN {X 0,Y 669.412,Z 830.209,A -85,B 0,C 180,E1 31079.312,E2 31079.312} C_VEL
LIN {X 0,Y 668.637,Z 851.268,A -85,B 0,C 180,E1 31078.791,E2 31078.791} C_VEL
LIN {X 0,Y 667.58,Z 876.147,A -85,B 0,C 180,E1 31078.006,E2 31078.006} C_VEL
LIN {X 0,Y 666.567,Z 896.343,A -85,B 0,C 180,E1 31077.227,E2 31077.227} C_VEL
LIN {X 0,Y 665.397,Z 918.586,A -85,B 0,C 180,E1 31076.219,E2 31076.219} C_VEL
LIN {X 0,Y 664.103,Z 939.836,A -85,B 0,C 180,E1 31075.077,E2 31075.077} C_VEL
LIN {X 0,Y 662.887,Z 960.588,A -85,B 0,C 180,E1 31073.797,E2 31073.797} C_VEL
LIN {X 0,Y 661.615,Z 980.256,A -85,B 0,C 180,E1 31072.386,E2 31072.386} C_VEL
LIN {X 0,Y 660.491,Z 999.282,A -85,B 0,C 180,E1 31070.84,E2 31070.84} C_VEL
LIN {X 0,Y 659.423,Z 1016.662,A -85,B 0,C 180,E1 31069.211,E2 31069.211} C_VEL
LIN {X 0,Y 658.556,Z 1032.899,A -85,B 0,C 180,E1 31067.495,E2 31067.495} C_VEL
LIN {X 0,Y 657.759,Z 1047.647,A -85,B 0,C 180,E1 31065.699,E2 31065.699} C_VEL
LIN {X 0,Y 657.167,Z 1061.255,A -85,B 0,C 180,E1 31063.82,E2 31063.82} C_VEL
LIN {X 0,Y 656.689,Z 1073.343,A -85,B 0,C 180,E1 31061.862,E2 31061.862} C_VEL
LIN {X 0,Y 656.368,Z 1084.218,A -85,B 0,C 180,E1 31059.824,E2 31059.824} C_VEL
LIN {X 0,Y 656.134,Z 1093.104,A -85,B 0,C 180,E1 31057.795,E2 31057.795} C_VEL
LIN {X 0,Y 655.998,Z 1100.157,A -85,B 0,C 180,E1 31055.861,E2 31055.861} C_VEL
LIN {X 0,Y 655.934,Z 1106.129,A -85,B 0,C 180,E1 31053.758,E2 31053.758} C_VEL
LIN {X 0,Y 655.924,Z 1110.006,A -85,B 0,C 180,E1 31051.922,E2 31051.922} C_VEL
LIN {X 0,Y 655.914,Z 1113.029,A -85,B 0,C 180,E1 31049.825,E2 31049.825} C_VEL
LIN {X 0,Y 655.899,Z 1114.309,A -85,B 0,C 180,E1 31047.728,E2 31047.728} C_VEL
LIN {X 0,Y 655.908,Z 1114.211,A -85,B 0,C 180,E1 31045.804,E2 31045.804} C_VEL
LIN {X 0,Y 655.918,Z 1112.432,A -85,B 0,C 180,E1 31043.611,E2 31043.611} C_VEL
LIN {X 0,Y 655.927,Z 1109.595,A -85,B 0,C 180,E1 31041.762,E2 31041.762} C_VEL
LIN {X 0,Y 655.962,Z 1104.875,A -85,B 0,C 180,E1 31039.638,E2 31039.638} C_VEL
LIN {X 0,Y 656.037,Z 1098.584,A -85,B 0,C 180,E1 31037.59,E2 31037.59} C_VEL
LIN {X 0,Y 656.179,Z 1091.12,A -85,B 0,C 180,E1 31035.618,E2 31035.618} C_VEL
LIN {X 0,Y 656.432,Z 1081.431,A -85,B 0,C 180,E1 31033.542,E2 31033.542} C_VEL
LIN {X 0,Y 656.764,Z 1071.468,A -85,B 0,C 180,E1 31031.722,E2 31031.722} C_VEL
LIN {X 0,Y 657.307,Z 1057.922,A -85,B 0,C 180,E1 31029.613,E2 31029.613} C_VEL
LIN {X 0,Y 657.909,Z 1044.912,A -85,B 0,C 180,E1 31027.857,E2 31027.857} C_VEL
LIN {X 0,Y 658.733,Z 1029.079,A -85,B 0,C 180,E1 31025.996,E2 31025.996} C_VEL
LIN {X 0,Y 659.607,Z 1013.672,A -85,B 0,C 180,E1 31024.404,E2 31024.404} C_VEL
LIN {X 0,Y 660.743,Z 994.431,A -85,B 0,C 180,E1 31022.661,E2 31022.661} C_VEL
LIN {X 0,Y 661.836,Z 977.129,A -85,B 0,C 180,E1 31021.286,E2 31021.286} C_VEL
LIN {X 0,Y 663.139,Z 955.883,A -85,B 0,C 180,E1 31019.811,E2 31019.811} C_VEL
LIN {X 0,Y 664.288,Z 936.891,A -85,B 0,C 180,E1 31018.664,E2 31018.664} C_VEL
LIN {X 0,Y 665.649,Z 913.923,A -85,B 0,C 180,E1 31017.468,E2 31017.468} C_VEL
LIN {X 0,Y 666.714,Z 893.239,A -85,B 0,C 180,E1 31016.554,E2 31016.554} C_VEL
LIN {X 0,Y 667.879,Z 870.001,A -85,B 0,C 180,E1 31015.69,E2 31015.69} C_VEL
LIN {X 0,Y 668.77,Z 848.126,A -85,B 0,C 180,E1 31015.035,E2 31015.035} C_VEL
LIN {X 0,Y 669.589,Z 825.779,A -85,B 0,C 180,E1 31014.5,E2 31014.5} C_VEL
LIN {X 0,Y 670.25,Z 799.004,A -85,B 0,C 180,E1 31014.038,E2 31014.038} C_VEL
LIN {X 0,Y 673.088,Z 545.561,A -85,B 0,C 180,E1 31010.967,E2 31010.967} C_VEL
LIN {X 0,Y 674.198,Z 442.006,A -85,B 0,C 180,E1 31009.686,E2 31009.686} C_VEL
LIN {X 0,Y 660.93,Z 419.584,A -85,B 0,C 180,E1 31008.492,E2 31008.492} C_VEL
LIN {X 0,Y 658.271,Z 415.259,A -85,B 0,C 180,E1 31008.229,E2 31008.229} C_VEL
LIN {X 0,Y 656.646,Z 410.614,A -85,B 0,C 180,E1 31007.664,E2 31007.664} C_VEL
LIN {X 0,Y 656.654,Z 410.432,A -85,B 0,C 180,E1 31004.675,E2 31004.675} C_VEL
LIN {X 0,Y 656.611,Z 410.402,A -85,B 0,C 180,E1 31001.953,E2 31001.953} C_VEL
LIN {X 0,Y 656.677,Z 410.432,A -85,B 0,C 180,E1 30999.191,E2 30999.191} C_VEL
LIN {X 0,Y 656.627,Z 410.39,A -85,B 0,C 180,E1 30996.189,E2 30996.189} C_VEL
LIN {X 0,Y 656.636,Z 410.432,A -85,B 0,C 180,E1 30993.557,E2 30993.557} C_VEL
LIN {X 0,Y 656.672,Z 410.393,A -85,B 0,C 180,E1 30990.468,E2 30990.468} C_VEL
LIN {X 0,Y 656.637,Z 410.421,A -85,B 0,C 180,E1 30987.674,E2 30987.674} C_VEL
LIN {X 0,Y 656.711,Z 410.419,A -85,B 0,C 180,E1 30984.753,E2 30984.753} C_VEL
LIN {X 0,Y 656.645,Z 410.431,A -85,B 0,C 180,E1 30981.811,E2 30981.811} C_VEL
LIN {X 0,Y 656.697,Z 410.426,A -85,B 0,C 180,E1 30978.924,E2 30978.924} C_VEL
LIN {X 0,Y 656.656,Z 410.416,A -85,B 0,C 180,E1 30975.817,E2 30975.817} C_VEL
LIN {X 0,Y 656.694,Z 410.431,A -85,B 0,C 180,E1 30972.934,E2 30972.934} C_VEL
LIN {X 0,Y 656.67,Z 410.426,A -85,B 0,C 180,E1 30969.819,E2 30969.819} C_VEL
LIN {X 0,Y 656.704,Z 410.419,A -85,B 0,C 180,E1 30966.821,E2 30966.821} C_VEL
LIN {X 0,Y 656.673,Z 410.426,A -85,B 0,C 180,E1 30963.667,E2 30963.667} C_VEL
LIN {X 0,Y 656.708,Z 410.425,A -85,B 0,C 180,E1 30960.611,E2 30960.611} C_VEL
LIN {X 0,Y 656.678,Z 410.416,A -85,B 0,C 180,E1 30957.556,E2 30957.556} C_VEL
LIN {X 0,Y 656.703,Z 410.427,A -85,B 0,C 180,E1 30954.496,E2 30954.496} C_VEL
LIN {X 0,Y 656.684,Z 410.419,A -85,B 0,C 180,E1 30951.418,E2 30951.418} C_VEL
LIN {X 0,Y 656.698,Z 410.417,A -85,B 0,C 180,E1 30948.405,E2 30948.405} C_VEL
LIN {X 0,Y 656.691,Z 410.426,A -85,B 0,C 180,E1 30945.359,E2 30945.359} C_VEL
LIN {X 0,Y 656.694,Z 410.428,A -85,B 0,C 180,E1 30942.27,E2 30942.27} C_VEL
LIN {X 0,Y 656.694,Z 410.421,A -85,B 0,C 180,E1 30939.21,E2 30939.21} C_VEL
LIN {X 0,Y 656.69,Z 410.431,A -85,B 0,C 180,E1 30936.203,E2 30936.203} C_VEL
LIN {X 0,Y 656.699,Z 410.41,A -85,B 0,C 180,E1 30933.114,E2 30933.114} C_VEL
LIN {X 0,Y 656.685,Z 410.425,A -85,B 0,C 180,E1 30930.139,E2 30930.139} C_VEL
LIN {X 0,Y 656.707,Z 410.424,A -85,B 0,C 180,E1 30927.073,E2 30927.073} C_VEL
LIN {X 0,Y 656.676,Z 410.423,A -85,B 0,C 180,E1 30924.003,E2 30924.003} C_VEL
LIN {X 0,Y 656.71,Z 410.417,A -85,B 0,C 180,E1 30921.036,E2 30921.036} C_VEL
LIN {X 0,Y 656.669,Z 410.419,A -85,B 0,C 180,E1 30917.935,E2 30917.935} C_VEL
LIN {X 0,Y 656.706,Z 410.418,A -85,B 0,C 180,E1 30914.927,E2 30914.927} C_VEL
LIN {X 0,Y 656.721,Z 410.667,A -85,B 0,C 180,E1 30912.179,E2 30912.179} C_VEL
LIN {X 0,Y 663.367,Z 427.94,A -85,B 0,C 180,E1 30910.231,E2 30910.231} C_VEL
LIN {X 0,Y 668.801,Z 442.613,A -85,B 0,C 180,E1 30908.701,E2 30908.701} C_VEL
LIN {X 0,Y 668.544,Z 452.088,A -85,B 0,C 180,E1 30908.019,E2 30908.019} C_VEL
LIN {X 0,Y 674.232,Z 477.069,A -85,B 0,C 180,E1 30907.307,E2 30907.307} C_VEL
LIN {X 0,Y 671.501,Z 721.883,A -85,B 0,C 180,E1 30904.326,E2 30904.326} C_VEL
LIN {X 0,Y 670.164,Z 843.308,A -85,B 0,C 180,E1 30902.849,E2 30902.849} C_VEL
LIN {X 0,Y 669.462,Z 868.873,A -85,B 0,C 180,E1 30902.387,E2 30902.387} C_VEL
LIN {X 0,Y 668.689,Z 889.892,A -85,B 0,C 180,E1 30901.872,E2 30901.872} C_VEL
LIN {X 0,Y 667.728,Z 913.254,A -85,B 0,C 180,E1 30901.156,E2 30901.156} C_VEL
LIN {X 0,Y 666.671,Z 934.203,A -85,B 0,C 180,E1 30900.361,E2 30900.361} C_VEL
LIN {X 0,Y 665.63,Z 954.266,A -85,B 0,C 180,E1 30899.47,E2 30899.47} C_VEL
LIN {X 0,Y 664.255,Z 977.414,A -85,B 0,C 180,E1 30898.261,E2 30898.261} C_VEL
LIN {X 0,Y 663.095,Z 996.725,A -85,B 0,C 180,E1 30897.09,E2 30897.09} C_VEL
LIN {X 0,Y 661.775,Z 1018.001,A -85,B 0,C 180,E1 30895.603,E2 30895.603} C_VEL
LIN {X 0,Y 660.695,Z 1035.398,A -85,B 0,C 180,E1 30894.213,E2 30894.213} C_VEL
LIN {X 0,Y 659.551,Z 1054.603,A -85,B 0,C 180,E1 30892.46,E2 30892.46} C_VEL
LIN {X 0,Y 658.697,Z 1069.63,A -85,B 0,C 180,E1 30890.899,E2 30890.899} C_VEL
LIN {X 0,Y 657.854,Z 1085.819,A -85,B 0,C 180,E1 30888.982,E2 30888.982} C_VEL
LIN {X 0,Y 657.286,Z 1098.521,A -85,B 0,C 180,E1 30887.256,E2 30887.256} C_VEL
LIN {X 0,Y 656.746,Z 1111.969,A -85,B 0,C 180,E1 30885.146,E2 30885.146} C_VEL
LIN {X 0,Y 656.405,Z 1122.022,A -85,B 0,C 180,E1 30883.298,E2 30883.298} C_VEL
LIN {X 0,Y 656.145,Z 1131.833,A -85,B 0,C 180,E1 30881.159,E2 30881.159} C_VEL
LIN {X 0,Y 656.035,Z 1138.817,A -85,B 0,C 180,E1 30879.297,E2 30879.297} C_VEL
LIN {X 0,Y 655.947,Z 1145.244,A -85,B 0,C 180,E1 30877.181,E2 30877.181} C_VEL
LIN {X 0,Y 655.895,Z 1149.656,A -85,B 0,C 180,E1 30875.16,E2 30875.16} C_VEL
LIN {X 0,Y 655.901,Z 1152.462,A -85,B 0,C 180,E1 30873.321,E2 30873.321} C_VEL
LIN {X 0,Y 655.909,Z 1154.215,A -85,B 0,C 180,E1 30871.136,E2 30871.136} C_VEL
LIN {X 0,Y 655.885,Z 1154.328,A -85,B 0,C 180,E1 30869.301,E2 30869.301} C_VEL
LIN {X 0,Y 655.889,Z 1153.226,A -85,B 0,C 180,E1 30867.379,E2 30867.379} C_VEL
LIN {X 0,Y 655.907,Z 1150.291,A -85,B 0,C 180,E1 30865.19,E2 30865.19} C_VEL
LIN {X 0,Y 655.937,Z 1146.483,A -85,B 0,C 180,E1 30863.347,E2 30863.347} C_VEL
LIN {X 0,Y 655.991,Z 1140.634,A -85,B 0,C 180,E1 30861.233,E2 30861.233} C_VEL
LIN {X 0,Y 656.124,Z 1133.604,A -85,B 0,C 180,E1 30859.285,E2 30859.285} C_VEL
LIN {X 0,Y 656.323,Z 1125.528,A -85,B 0,C 180,E1 30857.417,E2 30857.417} C_VEL
LIN {X 0,Y 656.666,Z 1114.351,A -85,B 0,C 180,E1 30855.269,E2 30855.269} C_VEL
LIN {X 0,Y 657.071,Z 1103.391,A -85,B 0,C 180,E1 30853.467,E2 30853.467} C_VEL
LIN {X 0,Y 657.695,Z 1089.324,A -85,B 0,C 180,E1 30851.473,E2 30851.473} C_VEL
LIN {X 0,Y 658.406,Z 1075.305,A -85,B 0,C 180,E1 30849.742,E2 30849.742} C_VEL
LIN {X 0,Y 659.336,Z 1058.307,A -85,B 0,C 180,E1 30847.908,E2 30847.908} C_VEL
LIN {X 0,Y 660.248,Z 1042.797,A -85,B 0,C 180,E1 30846.434,E2 30846.434} C_VEL
LIN {X 0,Y 661.459,Z 1022.865,A -85,B 0,C 180,E1 30844.768,E2 30844.768} C_VEL
LIN {X 0,Y 662.618,Z 1004.407,A -85,B 0,C 180,E1 30843.423,E2 30843.423} C_VEL
LIN {X 0,Y 663.968,Z 982.358,A -85,B 0,C 180,E1 30842.024,E2 30842.024} C_VEL
LIN {X 0,Y 665.114,Z 962.745,A -85,B 0,C 180,E1 30840.949,E2 30840.949} C_VEL
LIN {X 0,Y 666.461,Z 938.728,A -85,B 0,C 180,E1 30839.828,E2 30839.828} C_VEL
LIN {X 0,Y 667.412,Z 919.676,A -85,B 0,C 180,E1 30839.078,E2 30839.078} C_VEL
LIN {X 0,Y 668.429,Z 897.141,A -85,B 0,C 180,E1 30838.328,E2 30838.328} C_VEL
LIN {X 0,Y 669.288,Z 873.179,A -85,B 0,C 180,E1 30837.708,E2 30837.708} C_VEL
LIN {X 0,Y 670.004,Z 850.869,A -85,B 0,C 180,E1 30837.268,E2 30837.268} C_VEL
LIN {X 0,Y 670.509,Z 817.947,A -85,B 0,C 180,E1 30836.825,E2 30836.825} C_VEL
LIN {X 0,Y 672.926,Z 587.172,A -85,B 0,C 180,E1 30834.039,E2 30834.039} C_VEL
LIN {X 0,Y 674.073,Z 475.589,A -85,B 0,C 180,E1 30832.663,E2 30832.663} C_VEL
LIN {X 0,Y 668.491,Z 451.581,A -85,B 0,C 180,E1 30831.957,E2 30831.957} C_VEL
LIN {X 0,Y 668.687,Z 441.952,A -85,B 0,C 180,E1 30831.236,E2 30831.236} C_VEL
LIN {X 0,Y 659.357,Z 417.508,A -85,B 0,C 180,E1 30828.647,E2 30828.647} C_VEL
LIN {X 0,Y 656.726,Z 410.737,A -85,B 0,C 180,E1 30827.876,E2 30827.876} C_VEL
LIN {X 0,Y 656.687,Z 410.434,A -85,B 0,C 180,E1 30826.831,E2 30826.831} C_VEL
LIN {X 0,Y 656.688,Z 410.428,A -85,B 0,C 180,E1 30823.803,E2 30823.803} C_VEL
LIN {X 0,Y 656.683,Z 410.395,A -85,B 0,C 180,E1 30820.669,E2 30820.669} C_VEL
LIN {X 0,Y 656.7,Z 410.426,A -85,B 0,C 180,E1 30817.63,E2 30817.63} C_VEL
LIN {X 0,Y 656.688,Z 410.428,A -85,B 0,C 180,E1 30814.501,E2 30814.501} C_VEL
LIN {X 0,Y 656.706,Z 410.429,A -85,B 0,C 180,E1 30811.483,E2 30811.483} C_VEL
LIN {X 0,Y 656.691,Z 410.413,A -85,B 0,C 180,E1 30808.348,E2 30808.348} C_VEL
LIN {X 0,Y 656.701,Z 410.42,A -85,B 0,C 180,E1 30805.254,E2 30805.254} C_VEL
LIN {X 0,Y 656.69,Z 410.424,A -85,B 0,C 180,E1 30802.186,E2 30802.186} C_VEL
